LIN {X -0.012,Y -443.315,Z 1451.571,A 0.000,B 0.000,C 90.000,E1 282.715} C_DIS
LIN {X -0.002,Y -444.816,Z 1451.568,A 0.000,B 0.000,C 90.000,E1 282.187} C_DIS
LIN {X 0.020,Y -445.994,Z 1451.565,A 0.000,B 0.000,C 90.000,E1 281.658} C_DIS
LIN {X 0.049,Y -446.747,Z 1451.562,A 0.000,B 0.000,C 90.000,E1 281.130} C_DIS
LIN {X 0.083,Y -447.090,Z 1451.559,A 0.000,B 0.000,C 90.000,E1 280.602} C_DIS
LIN {X 0.118,Y -446.958,Z 1451.556,A 0.000,B 0.000,C 90.000,E1 280.074} C_DIS
LIN {X 0.078,Y -446.263,Z 1451.553,A 0.000,B 0.000,C 90.000,E1 279.557} C_DIS
LIN {X 0.112,Y -445.021,Z 1451.550,A 0.000,B 0.000,C 90.000,E1 279.029} C_DIS
LIN {X 0.071,Y -443.207,Z 1451.547,A 0.000,B 0.000,C 90.000,E1 278.511} C_DIS
LIN {X 0.025,Y -440.657,Z 1451.544,A 0.000,B 0.000,C 90.000,E1 277.992} C_DIS
LIN {X 0.022,Y -437.241,Z 1451.542,A 0.000,B 0.000,C 90.000,E1 277.466} C_DIS
LIN {X -0.056,Y -432.786,Z 1451.539,A 0.000,B 0.000,C 90.000,E1 276.947} C_DIS
LIN {X -0.155,Y -427.058,Z 1451.536,A 0.000,B 0.000,C 90.000,E1 276.429} C_DIS
LIN {X 0.194,Y -420.712,Z 1451.533,A 0.000,B 0.000,C 90.000,E1 275.910} C_DIS
LIN {X 0.170,Y -414.293,Z 1451.531,A 0.000,B 0.000,C 90.000,E1 275.511} C_DIS
LIN {X 0.133,Y -407.868,Z 1451.529,A 0.000,B 0.000,C 90.000,E1 275.163} C_DIS
LIN {X 0.107,Y -397.871,Z 1451.526,A 0.000,B 0.000,C 90.000,E1 274.702} C_DIS
LIN {X 0.086,Y -388.083,Z 1451.524,A 0.000,B 0.000,C 90.000,E1 274.302} C_DIS
LIN {X 0.003,Y -369.176,Z 1451.520,A 0.000,B 0.000,C 90.000,E1 273.612} C_DIS
LIN {X 0.038,Y -359.489,Z 1451.518,A 0.000,B 0.000,C 90.000,E1 273.269} C_DIS
LIN {X -0.062,Y -349.143,Z 1451.516,A 0.000,B 0.000,C 90.000,E1 272.980} C_DIS
LIN {X 0.134,Y -338.896,Z 1451.515,A 0.000,B 0.000,C 90.000,E1 272.694} C_DIS
LIN {X -0.136,Y -327.379,Z 1451.514,A 0.000,B 0.000,C 90.000,E1 272.522} C_DIS
LIN {X -0.109,Y -314.439,Z 1451.513,A 0.000,B 0.000,C 90.000,E1 272.350} C_DIS
LIN {X 0.000,Y -302.497,Z 1451.512,A 0.000,B 0.000,C 90.000,E1 272.236} C_DIS
LIN {X -0.035,Y -181.227,Z 1451.512,A 0.000,B 0.000,C 90.000,E1 272.236} C_DIS
LIN {X -0.026,Y -181.564,Z 1451.503,A 0.000,B 0.000,C 90.000,E1 270.516} C_DIS
LIN {X -0.036,Y -181.121,Z 1451.489,A 0.000,B 0.000,C 90.000,E1 267.993} C_DIS
LIN {X -0.047,Y -180.907,Z 1451.475,A 0.000,B 0.000,C 90.000,E1 265.469} C_DIS
LIN {X 0.009,Y -180.730,Z 1451.470,A 0.000,B 0.000,C 90.000,E1 264.609} C_DIS
LIN {X -0.069,Y -178.819,Z 1451.442,A 0.000,B 0.000,C 90.000,E1 259.567} C_DIS
LIN {X 0.013,Y -175.863,Z 1451.414,A 0.000,B 0.000,C 90.000,E1 254.448} C_DIS
LIN {X 0.062,Y -173.831,Z 1451.399,A 0.000,B 0.000,C 90.000,E1 251.873} C_DIS
LIN {X -0.003,Y -171.498,Z 1451.380,A 0.000,B 0.000,C 90.000,E1 248.465} C_DIS
LIN {X -0.017,Y -167.726,Z 1451.356,A 0.000,B 0.000,C 90.000,E1 244.152} C_DIS
LIN {X 0.000,Y -166.421,Z 1451.347,A 0.000,B 0.000,C 90.000,E1 242.410} C_DIS
LIN {X -0.002,Y -163.142,Z 1451.327,A 0.000,B 0.000,C 90.000,E1 238.918} C_DIS
LIN {X -0.036,Y -161.097,Z 1451.313,A 0.000,B 0.000,C 90.000,E1 236.294} C_DIS
LIN {X -0.052,Y -157.825,Z 1451.293,A 0.000,B 0.000,C 90.000,E1 232.763} C_DIS
LIN {X 0.011,Y -155.859,Z 1451.278,A 0.000,B 0.000,C 90.000,E1 230.070} C_DIS
LIN {X 0.067,Y -152.108,Z 1451.253,A 0.000,B 0.000,C 90.000,E1 225.567} C_DIS
LIN {X -0.026,Y -150.359,Z 1451.238,A 0.000,B 0.000,C 90.000,E1 222.894} C_DIS
LIN {X 0.013,Y -147.094,Z 1451.213,A 0.000,B 0.000,C 90.000,E1 218.338} C_DIS
LIN {X 0.008,Y -145.665,Z 1451.198,A 0.000,B 0.000,C 90.000,E1 215.598} C_DIS
LIN {X 0.012,Y -143.047,Z 1451.172,A 0.000,B 0.000,C 90.000,E1 211.003} C_DIS
LIN {X 0.012,Y -141.671,Z 1451.152,A 0.000,B 0.000,C 90.000,E1 207.308} C_DIS
LIN {X 0.057,Y -139.452,Z 1451.116,A 0.000,B 0.000,C 90.000,E1 200.791} C_DIS
LIN {X -0.023,Y -139.186,Z 1451.105,A 0.000,B 0.000,C 90.000,E1 198.960} C_DIS
LIN {X 0.000,Y -138.322,Z 1451.053,A 0.000,B 0.000,C 90.000,E1 189.613} C_DIS
LIN {X 0.007,Y -139.460,Z 1451.007,A 0.000,B 0.000,C 90.000,E1 181.203} C_DIS
LIN {X -0.053,Y -141.016,Z 1450.976,A 0.000,B 0.000,C 90.000,E1 175.641} C_DIS
LIN {X 0.037,Y -142.770,Z 1450.955,A 0.000,B 0.000,C 90.000,E1 171.894} C_DIS
LIN {X -0.007,Y -145.180,Z 1450.929,A 0.000,B 0.000,C 90.000,E1 167.297} C_DIS
LIN {X 0.026,Y -147.802,Z 1450.909,A 0.000,B 0.000,C 90.000,E1 163.614} C_DIS
LIN {X -0.079,Y -150.488,Z 1450.889,A 0.000,B 0.000,C 90.000,E1 160.007} C_DIS
LIN {X -0.007,Y -153.944,Z 1450.869,A 0.000,B 0.000,C 90.000,E1 156.357} C_DIS
LIN {X 0.057,Y -157.355,Z 1450.849,A 0.000,B 0.000,C 90.000,E1 152.743} C_DIS
LIN {X 0.000,Y -161.551,Z 1450.829,A 0.000,B 0.000,C 90.000,E1 149.203} C_DIS
LIN {X 0.013,Y -165.750,Z 1450.809,A 0.000,B 0.000,C 90.000,E1 145.674} C_DIS
LIN {X 0.000,Y -170.704,Z 1450.790,A 0.000,B 0.000,C 90.000,E1 142.190} C_DIS
LIN {X -0.089,Y -175.578,Z 1450.771,A 0.000,B 0.000,C 90.000,E1 138.771} C_DIS
LIN {X 0.030,Y -181.195,Z 1450.752,A 0.000,B 0.000,C 90.000,E1 135.324} C_DIS
LIN {X 0.023,Y -186.657,Z 1450.733,A 0.000,B 0.000,C 90.000,E1 131.962} C_DIS
LIN {X -0.032,Y -191.261,Z 1450.719,A 0.000,B 0.000,C 90.000,E1 129.483} C_DIS
LIN {X 0.048,Y -197.082,Z 1450.701,A 0.000,B 0.000,C 90.000,E1 126.171} C_DIS
LIN {X 0.036,Y -200.634,Z 1450.691,A 0.000,B 0.000,C 90.000,E1 124.405} C_DIS
LIN {X 0.020,Y -312.743,Z 1450.691,A 0.000,B 0.000,C 90.000,E1 124.405} C_DIS
LIN {X 0.046,Y -314.887,Z 1450.691,A 0.000,B 0.000,C 90.000,E1 124.358} C_DIS
LIN {X -0.085,Y -320.371,Z 1450.689,A 0.000,B 0.000,C 90.000,E1 124.072} C_DIS
LIN {X -0.040,Y -323.325,Z 1450.688,A 0.000,B 0.000,C 90.000,E1 123.754} C_DIS
LIN {X 0.032,Y -325.329,Z 1450.686,A 0.000,B 0.000,C 90.000,E1 123.452} C_DIS
LIN {X 0.015,Y -326.896,Z 1450.684,A 0.000,B 0.000,C 90.000,E1 123.166} C_DIS
LIN {X -0.061,Y -329.384,Z 1450.681,A 0.000,B 0.000,C 90.000,E1 122.546} C_DIS
LIN {X -0.136,Y -340.169,Z 1450.665,A 0.000,B 0.000,C 90.000,E1 119.745} C_DIS
LIN {X 0.067,Y -352.322,Z 1450.650,A 0.000,B 0.000,C 90.000,E1 116.950} C_DIS
LIN {X -0.017,Y -365.945,Z 1450.635,A 0.000,B 0.000,C 90.000,E1 114.259} C_DIS
LIN {X 0.042,Y -379.384,Z 1450.622,A 0.000,B 0.000,C 90.000,E1 111.897} C_DIS
LIN {X 0.170,Y -394.173,Z 1450.609,A 0.000,B 0.000,C 90.000,E1 109.577} C_DIS
LIN {X 0.040,Y -410.411,Z 1450.596,A 0.000,B 0.000,C 90.000,E1 107.347} C_DIS
LIN {X -0.222,Y -428.214,Z 1450.584,A 0.000,B 0.000,C 90.000,E1 105.190} C_DIS
LIN {X -0.210,Y -447.601,Z 1450.572,A 0.000,B 0.000,C 90.000,E1 103.063} C_DIS
LIN {X -0.068,Y -467.784,Z 1450.562,A 0.000,B 0.000,C 90.000,E1 101.074} C_DIS
LIN {X -0.089,Y -488.295,Z 1450.551,A 0.000,B 0.000,C 90.000,E1 99.265} C_DIS
LIN {X 0.066,Y -490.122,Z 1450.550,A 0.000,B 0.000,C 90.000,E1 99.029} C_DIS
LIN {X -0.110,Y -491.699,Z 1450.549,A 0.000,B 0.000,C 90.000,E1 98.803} C_DIS
LIN {X -0.211,Y -492.876,Z 1450.547,A 0.000,B 0.000,C 90.000,E1 98.568} C_DIS
LIN {X 0.020,Y -494.284,Z 1450.545,A 0.000,B 0.000,C 90.000,E1 98.049} C_DIS
LIN {X -0.229,Y -494.640,Z 1450.542,A 0.000,B 0.000,C 90.000,E1 97.587} C_DIS
LIN {X 0.022,Y -494.007,Z 1450.539,A 0.000,B 0.000,C 90.000,E1 97.068} C_DIS
LIN {X -0.215,Y -492.279,Z 1450.537,A 0.000,B 0.000,C 90.000,E1 96.606} C_DIS
LIN {X 0.180,Y -490.905,Z 1450.535,A 0.000,B 0.000,C 90.000,E1 96.315} C_DIS
LIN {X 0.168,Y -479.194,Z 1450.526,A 0.000,B 0.000,C 90.000,E1 94.588} C_DIS
LIN {X -0.108,Y -468.504,Z 1450.516,A 0.000,B 0.000,C 90.000,E1 92.865} C_DIS
LIN {X -0.173,Y -460.284,Z 1450.509,A 0.000,B 0.000,C 90.000,E1 91.604} C_DIS
LIN {X -0.173,Y -446.693,Z 1450.497,A 0.000,B 0.000,C 90.000,E1 89.542} C_DIS
LIN {X -0.032,Y -433.500,Z 1450.486,A 0.000,B 0.000,C 90.000,E1 87.421} C_DIS
LIN {X 0.123,Y -421.927,Z 1450.475,A 0.000,B 0.000,C 90.000,E1 85.527} C_DIS
LIN {X 0.073,Y -410.380,Z 1450.465,A 0.000,B 0.000,C 90.000,E1 83.628} C_DIS
LIN {X -0.173,Y -398.612,Z 1450.454,A 0.000,B 0.000,C 90.000,E1 81.724} C_DIS
LIN {X -0.138,Y -386.759,Z 1450.443,A 0.000,B 0.000,C 90.000,E1 79.746} C_DIS
LIN {X 0.106,Y -373.467,Z 1450.430,A 0.000,B 0.000,C 90.000,E1 77.409} C_DIS
LIN {X 0.123,Y -362.107,Z 1450.419,A 0.000,B 0.000,C 90.000,E1 75.353} C_DIS
LIN {X 0.085,Y -350.791,Z 1450.407,A 0.000,B 0.000,C 90.000,E1 73.268} C_DIS
LIN {X 0.017,Y -339.368,Z 1450.395,A 0.000,B 0.000,C 90.000,E1 71.148} C_DIS
LIN {X 0.116,Y -326.454,Z 1450.381,A 0.000,B 0.000,C 90.000,E1 68.646} C_DIS
LIN {X 0.065,Y -312.613,Z 1450.366,A 0.000,B 0.000,C 90.000,E1 65.793} C_DIS
LIN {X -0.090,Y -296.897,Z 1450.346,A 0.000,B 0.000,C 90.000,E1 62.231} C_DIS
LIN {X -0.034,Y -283.966,Z 1450.327,A 0.000,B 0.000,C 90.000,E1 58.869} C_DIS
LIN {X -0.109,Y -273.172,Z 1450.310,A 0.000,B 0.000,C 90.000,E1 55.801} C_DIS
LIN {X 0.034,Y -261.705,Z 1450.290,A 0.000,B 0.000,C 90.000,E1 52.271} C_DIS
LIN {X 0.069,Y -251.127,Z 1450.271,A 0.000,B 0.000,C 90.000,E1 48.690} C_DIS
LIN {X -0.076,Y -241.586,Z 1450.250,A 0.000,B 0.000,C 90.000,E1 45.081} C_DIS
LIN {X -0.007,Y -232.924,Z 1450.230,A 0.000,B 0.000,C 90.000,E1 41.353} C_DIS
LIN {X 0.022,Y -225.169,Z 1450.209,A 0.000,B 0.000,C 90.000,E1 37.569} C_DIS
LIN {X 0.120,Y -218.260,Z 1450.187,A 0.000,B 0.000,C 90.000,E1 33.706} C_DIS
LIN {X -0.101,Y -212.091,Z 1450.166,A 0.000,B 0.000,C 90.000,E1 29.873} C_DIS
LIN {X 0.016,Y -206.777,Z 1450.144,A 0.000,B 0.000,C 90.000,E1 25.899} C_DIS
LIN {X 0.071,Y -202.307,Z 1450.122,A 0.000,B 0.000,C 90.000,E1 21.897} C_DIS
LIN {X -0.033,Y -197.929,Z 1450.095,A 0.000,B 0.000,C 90.000,E1 17.094} C_DIS
LIN {X 0.071,Y -194.655,Z 1450.068,A 0.000,B 0.000,C 90.000,E1 12.187} C_DIS
LIN {X 0.043,Y -192.713,Z 1450.045,A 0.000,B 0.000,C 90.000,E1 8.106} C_DIS
LIN {X 0.053,Y -190.911,Z 1450.013,A 0.000,B 0.000,C 90.000,E1 2.350} C_DIS
LIN {X 0.010,Y -190.278,Z 1449.988,A 0.000,B 0.000,C 90.000,E1 357.879} C_DIS
LIN {X -0.079,Y -190.435,Z 1449.956,A 0.000,B 0.000,C 90.000,E1 352.129} C_DIS
LIN {X -0.059,Y -191.810,Z 1449.924,A 0.000,B 0.000,C 90.000,E1 346.353} C_DIS
LIN {X -0.056,Y -194.696,Z 1449.892,A 0.000,B 0.000,C 90.000,E1 340.604} C_DIS
LIN {X 0.105,Y -198.511,Z 1449.865,A 0.000,B 0.000,C 90.000,E1 335.665} C_DIS
LIN {X 0.039,Y -202.895,Z 1449.843,A 0.000,B 0.000,C 90.000,E1 331.641} C_DIS
LIN {X -0.042,Y -208.476,Z 1449.820,A 0.000,B 0.000,C 90.000,E1 327.661} C_DIS
LIN {X 0.003,Y -213.898,Z 1449.803,A 0.000,B 0.000,C 90.000,E1 324.482} C_DIS
LIN {X 0.088,Y -220.301,Z 1449.785,A 0.000,B 0.000,C 90.000,E1 321.331} C_DIS
LIN {X 0.039,Y -228.594,Z 1449.766,A 0.000,B 0.000,C 90.000,E1 317.877} C_DIS
LIN {X -0.120,Y -238.107,Z 1449.747,A 0.000,B 0.000,C 90.000,E1 314.514} C_DIS
LIN {X 0.017,Y -247.599,Z 1449.731,A 0.000,B 0.000,C 90.000,E1 311.515} C_DIS
LIN {X -0.026,Y -259.668,Z 1449.713,A 0.000,B 0.000,C 90.000,E1 308.257} C_DIS
LIN {X 0.028,Y -270.155,Z 1449.699,A 0.000,B 0.000,C 90.000,E1 305.758} C_DIS
LIN {X 0.067,Y -280.287,Z 1449.687,A 0.000,B 0.000,C 90.000,E1 303.658} C_DIS
LIN {X 0.017,Y -289.691,Z 1449.678,A 0.000,B 0.000,C 90.000,E1 301.957} C_DIS
LIN {X 0.108,Y -300.162,Z 1449.668,A 0.000,B 0.000,C 90.000,E1 300.256} C_DIS
LIN {X 0.028,Y -309.441,Z 1449.661,A 0.000,B 0.000,C 90.000,E1 298.949} C_DIS
LIN {X -0.048,Y -319.596,Z 1449.654,A 0.000,B 0.000,C 90.000,E1 297.692} C_DIS
LIN {X -0.052,Y -335.747,Z 1449.644,A 0.000,B 0.000,C 90.000,E1 295.899} C_DIS
LIN {X -0.142,Y -349.504,Z 1449.636,A 0.000,B 0.000,C 90.000,E1 294.515} C_DIS
LIN {X 0.040,Y -362.886,Z 1449.629,A 0.000,B 0.000,C 90.000,E1 293.131} C_DIS
LIN {X -0.080,Y -373.257,Z 1449.623,A 0.000,B 0.000,C 90.000,E1 292.078} C_DIS
LIN {X 0.040,Y -386.282,Z 1449.615,A 0.000,B 0.000,C 90.000,E1 290.663} C_DIS
LIN {X -0.199,Y -396.420,Z 1449.609,A 0.000,B 0.000,C 90.000,E1 289.577} C_DIS
LIN {X 0.146,Y -408.840,Z 1449.601,A 0.000,B 0.000,C 90.000,E1 288.127} C_DIS
LIN {X -0.081,Y -416.029,Z 1449.596,A 0.000,B 0.000,C 90.000,E1 287.330} C_DIS
LIN {X 0.001,Y -422.783,Z 1449.592,A 0.000,B 0.000,C 90.000,E1 286.496} C_DIS
LIN {X 0.155,Y -428.836,Z 1449.587,A 0.000,B 0.000,C 90.000,E1 285.662} C_DIS
LIN {X -0.168,Y -433.987,Z 1449.583,A 0.000,B 0.000,C 90.000,E1 284.898} C_DIS
LIN {X 0.092,Y -438.179,Z 1449.578,A 0.000,B 0.000,C 90.000,E1 284.064} C_DIS
LIN {X 0.074,Y -440.546,Z 1449.575,A 0.000,B 0.000,C 90.000,E1 283.536} C_DIS
LIN {X -0.143,Y -443.448,Z 1449.571,A 0.000,B 0.000,C 90.000,E1 282.771} C_DIS
LIN {X -0.133,Y -444.982,Z 1449.568,A 0.000,B 0.000,C 90.000,E1 282.243} C_DIS
LIN {X -0.112,Y -446.197,Z 1449.565,A 0.000,B 0.000,C 90.000,E1 281.715} C_DIS
LIN {X -0.083,Y -447.028,Z 1449.562,A 0.000,B 0.000,C 90.000,E1 281.186} C_DIS
LIN {X -0.049,Y -447.415,Z 1449.559,A 0.000,B 0.000,C 90.000,E1 280.658} C_DIS
LIN {X -0.092,Y -447.295,Z 1449.556,A 0.000,B 0.000,C 90.000,E1 280.141} C_DIS
LIN {X -0.052,Y -446.719,Z 1449.553,A 0.000,B 0.000,C 90.000,E1 279.613} C_DIS
LIN {X -0.087,Y -445.545,Z 1449.550,A 0.000,B 0.000,C 90.000,E1 279.095} C_DIS
LIN {X -0.055,Y -443.776,Z 1449.548,A 0.000,B 0.000,C 90.000,E1 278.568} C_DIS
LIN {X -0.097,Y -441.304,Z 1449.545,A 0.000,B 0.000,C 90.000,E1 278.049} C_DIS
LIN {X -0.153,Y -437.981,Z 1449.542,A 0.000,B 0.000,C 90.000,E1 277.530} C_DIS
LIN {X -0.170,Y -433.708,Z 1449.539,A 0.000,B 0.000,C 90.000,E1 277.004} C_DIS
LIN {X 0.163,Y -428.146,Z 1449.536,A 0.000,B 0.000,C 90.000,E1 276.429} C_DIS
LIN {X -0.017,Y -421.798,Z 1449.533,A 0.000,B 0.000,C 90.000,E1 275.967} C_DIS
LIN {X -0.118,Y -415.309,Z 1449.531,A 0.000,B 0.000,C 90.000,E1 275.568} C_DIS
LIN {X -0.198,Y -408.819,Z 1449.529,A 0.000,B 0.000,C 90.000,E1 275.220} C_DIS
LIN {X -0.046,Y -402.223,Z 1449.527,A 0.000,B 0.000,C 90.000,E1 274.878} C_DIS
LIN {X -0.152,Y -392.450,Z 1449.525,A 0.000,B 0.000,C 90.000,E1 274.473} C_DIS
LIN {X 0.004,Y -379.550,Z 1449.522,A 0.000,B 0.000,C 90.000,E1 273.955} C_DIS
LIN {X 0.027,Y -363.639,Z 1449.519,A 0.000,B 0.000,C 90.000,E1 273.383} C_DIS
LIN {X -0.123,Y -353.816,Z 1449.517,A 0.000,B 0.000,C 90.000,E1 273.094} C_DIS
LIN {X 0.163,Y -339.985,Z 1449.515,A 0.000,B 0.000,C 90.000,E1 272.694} C_DIS
LIN {X -0.039,Y -332.780,Z 1449.514,A 0.000,B 0.000,C 90.000,E1 272.579} C_DIS
LIN {X -0.099,Y -320.374,Z 1449.513,A 0.000,B 0.000,C 90.000,E1 272.407} C_DIS
LIN {X -0.029,Y -310.790,Z 1449.513,A 0.000,B 0.000,C 90.000,E1 272.293} C_DIS
LIN {X -0.021,Y -301.329,Z 1449.512,A 0.000,B 0.000,C 90.000,E1 272.236} C_DIS
LIN {X -0.048,Y -181.227,Z 1449.512,A 0.000,B 0.000,C 90.000,E1 272.236} C_DIS
LIN {X -0.007,Y -181.563,Z 1449.503,A 0.000,B 0.000,C 90.000,E1 270.516} C_DIS
LIN {X -0.077,Y -181.281,Z 1449.494,A 0.000,B 0.000,C 90.000,E1 268.854} C_DIS
LIN {X -0.028,Y -180.906,Z 1449.475,A 0.000,B 0.000,C 90.000,E1 265.469} C_DIS
LIN {X 0.029,Y -180.733,Z 1449.470,A 0.000,B 0.000,C 90.000,E1 264.609} C_DIS
LIN {X -0.050,Y -178.821,Z 1449.442,A 0.000,B 0.000,C 90.000,E1 259.567} C_DIS
LIN {X 0.032,Y -175.866,Z 1449.414,A 0.000,B 0.000,C 90.000,E1 254.448} C_DIS
LIN {X 0.027,Y -173.835,Z 1449.399,A 0.000,B 0.000,C 90.000,E1 251.891} C_DIS
LIN {X 0.016,Y -171.504,Z 1449.380,A 0.000,B 0.000,C 90.000,E1 248.465} C_DIS
LIN {X 0.003,Y -167.731,Z 1449.356,A 0.000,B 0.000,C 90.000,E1 244.152} C_DIS
LIN {X 0.018,Y -166.427,Z 1449.347,A 0.000,B 0.000,C 90.000,E1 242.410} C_DIS
LIN {X 0.016,Y -163.148,Z 1449.327,A 0.000,B 0.000,C 90.000,E1 238.918} C_DIS
LIN {X -0.018,Y -161.103,Z 1449.313,A 0.000,B 0.000,C 90.000,E1 236.294} C_DIS
LIN {X -0.035,Y -157.830,Z 1449.293,A 0.000,B 0.000,C 90.000,E1 232.763} C_DIS
LIN {X 0.029,Y -155.864,Z 1449.278,A 0.000,B 0.000,C 90.000,E1 230.070} C_DIS
LIN {X 0.084,Y -152.113,Z 1449.253,A 0.000,B 0.000,C 90.000,E1 225.567} C_DIS
LIN {X -0.008,Y -150.363,Z 1449.238,A 0.000,B 0.000,C 90.000,E1 222.894} C_DIS
LIN {X 0.030,Y -147.099,Z 1449.213,A 0.000,B 0.000,C 90.000,E1 218.338} C_DIS
LIN {X 0.025,Y -145.668,Z 1449.198,A 0.000,B 0.000,C 90.000,E1 215.598} C_DIS
LIN {X 0.028,Y -143.051,Z 1449.172,A 0.000,B 0.000,C 90.000,E1 211.003} C_DIS
LIN {X -0.036,Y -141.673,Z 1449.152,A 0.000,B 0.000,C 90.000,E1 207.334} C_DIS
LIN {X 0.072,Y -139.453,Z 1449.116,A 0.000,B 0.000,C 90.000,E1 200.791} C_DIS
LIN {X -0.007,Y -139.187,Z 1449.105,A 0.000,B 0.000,C 90.000,E1 198.960} C_DIS
LIN {X 0.016,Y -138.322,Z 1449.053,A 0.000,B 0.000,C 90.000,E1 189.613} C_DIS
LIN {X 0.023,Y -139.459,Z 1449.007,A 0.000,B 0.000,C 90.000,E1 181.203} C_DIS
LIN {X -0.036,Y -141.013,Z 1448.976,A 0.000,B 0.000,C 90.000,E1 175.641} C_DIS
LIN {X 0.054,Y -142.767,Z 1448.955,A 0.000,B 0.000,C 90.000,E1 171.894} C_DIS
LIN {X 0.009,Y -145.176,Z 1448.929,A 0.000,B 0.000,C 90.000,E1 167.297} C_DIS
LIN {X 0.042,Y -147.798,Z 1448.909,A 0.000,B 0.000,C 90.000,E1 163.614} C_DIS
LIN {X -0.062,Y -150.482,Z 1448.889,A 0.000,B 0.000,C 90.000,E1 160.007} C_DIS
LIN {X 0.011,Y -153.937,Z 1448.869,A 0.000,B 0.000,C 90.000,E1 156.357} C_DIS
LIN {X 0.075,Y -157.348,Z 1448.849,A 0.000,B 0.000,C 90.000,E1 152.743} C_DIS
LIN {X 0.018,Y -161.543,Z 1448.829,A 0.000,B 0.000,C 90.000,E1 149.203} C_DIS
LIN {X 0.030,Y -165.742,Z 1448.809,A 0.000,B 0.000,C 90.000,E1 145.674} C_DIS
LIN {X 0.018,Y -170.694,Z 1448.790,A 0.000,B 0.000,C 90.000,E1 142.190} C_DIS
LIN {X -0.071,Y -175.568,Z 1448.771,A 0.000,B 0.000,C 90.000,E1 138.771} C_DIS
LIN {X 0.049,Y -181.186,Z 1448.752,A 0.000,B 0.000,C 90.000,E1 135.324} C_DIS
LIN {X -0.082,Y -186.646,Z 1448.733,A 0.000,B 0.000,C 90.000,E1 132.000} C_DIS
LIN {X -0.013,Y -191.252,Z 1448.719,A 0.000,B 0.000,C 90.000,E1 129.483} C_DIS
LIN {X 0.068,Y -197.071,Z 1448.701,A 0.000,B 0.000,C 90.000,E1 126.171} C_DIS
LIN {X -0.031,Y -200.580,Z 1448.691,A 0.000,B 0.000,C 90.000,E1 124.452} C_DIS
LIN {X 0.158,Y -312.400,Z 1448.691,A 0.000,B 0.000,C 90.000,E1 124.405} C_DIS
LIN {X -0.080,Y -317.681,Z 1448.690,A 0.000,B 0.000,C 90.000,E1 124.278} C_DIS
LIN {X -0.144,Y -320.108,Z 1448.689,A 0.000,B 0.000,C 90.000,E1 124.119} C_DIS
LIN {X -0.188,Y -323.361,Z 1448.688,A 0.000,B 0.000,C 90.000,E1 123.785} C_DIS
LIN {X 0.066,Y -325.332,Z 1448.686,A 0.000,B 0.000,C 90.000,E1 123.452} C_DIS
LIN {X 0.049,Y -326.878,Z 1448.684,A 0.000,B 0.000,C 90.000,E1 123.166} C_DIS
LIN {X -0.025,Y -329.341,Z 1448.681,A 0.000,B 0.000,C 90.000,E1 122.546} C_DIS
LIN {X -0.102,Y -340.123,Z 1448.665,A 0.000,B 0.000,C 90.000,E1 119.745} C_DIS
LIN {X 0.101,Y -352.275,Z 1448.650,A 0.000,B 0.000,C 90.000,E1 116.950} C_DIS
LIN {X 0.017,Y -365.892,Z 1448.635,A 0.000,B 0.000,C 90.000,E1 114.259} C_DIS
LIN {X 0.076,Y -379.329,Z 1448.622,A 0.000,B 0.000,C 90.000,E1 111.897} C_DIS
LIN {X -0.168,Y -394.114,Z 1448.609,A 0.000,B 0.000,C 90.000,E1 109.631} C_DIS
LIN {X 0.074,Y -410.349,Z 1448.596,A 0.000,B 0.000,C 90.000,E1 107.347} C_DIS
LIN {X -0.188,Y -428.149,Z 1448.584,A 0.000,B 0.000,C 90.000,E1 105.190} C_DIS
LIN {X -0.176,Y -447.532,Z 1448.572,A 0.000,B 0.000,C 90.000,E1 103.063} C_DIS
LIN {X -0.037,Y -467.715,Z 1448.562,A 0.000,B 0.000,C 90.000,E1 101.074} C_DIS
LIN {X -0.216,Y -485.820,Z 1448.553,A 0.000,B 0.000,C 90.000,E1 99.500} C_DIS
LIN {X -0.061,Y -488.216,Z 1448.551,A 0.000,B 0.000,C 90.000,E1 99.265} C_DIS
LIN {X 0.094,Y -490.036,Z 1448.550,A 0.000,B 0.000,C 90.000,E1 99.029} C_DIS
LIN {X -0.082,Y -491.607,Z 1448.549,A 0.000,B 0.000,C 90.000,E1 98.803} C_DIS
LIN {X -0.183,Y -492.779,Z 1448.547,A 0.000,B 0.000,C 90.000,E1 98.568} C_DIS
LIN {X 0.048,Y -494.181,Z 1448.545,A 0.000,B 0.000,C 90.000,E1 98.049} C_DIS
LIN {X -0.201,Y -494.532,Z 1448.542,A 0.000,B 0.000,C 90.000,E1 97.587} C_DIS
LIN {X 0.048,Y -493.891,Z 1448.539,A 0.000,B 0.000,C 90.000,E1 97.068} C_DIS
LIN {X -0.189,Y -492.157,Z 1448.537,A 0.000,B 0.000,C 90.000,E1 96.606} C_DIS
LIN {X 0.206,Y -490.779,Z 1448.535,A 0.000,B 0.000,C 90.000,E1 96.315} C_DIS
LIN {X 0.190,Y -479.064,Z 1448.526,A 0.000,B 0.000,C 90.000,E1 94.588} C_DIS
LIN {X -0.090,Y -468.330,Z 1448.516,A 0.000,B 0.000,C 90.000,E1 92.865} C_DIS
LIN {X -0.156,Y -460.116,Z 1448.509,A 0.000,B 0.000,C 90.000,E1 91.604} C_DIS
LIN {X -0.161,Y -446.531,Z 1448.497,A 0.000,B 0.000,C 90.000,E1 89.542} C_DIS
LIN {X -0.023,Y -433.380,Z 1448.486,A 0.000,B 0.000,C 90.000,E1 87.421} C_DIS
LIN {X 0.128,Y -421.841,Z 1448.475,A 0.000,B 0.000,C 90.000,E1 85.527} C_DIS
LIN {X 0.077,Y -410.317,Z 1448.465,A 0.000,B 0.000,C 90.000,E1 83.628} C_DIS
LIN {X 0.197,Y -400.277,Z 1448.455,A 0.000,B 0.000,C 90.000,E1 81.951} C_DIS
LIN {X 0.136,Y -390.147,Z 1448.446,A 0.000,B 0.000,C 90.000,E1 80.274} C_DIS
LIN {X 0.095,Y -375.153,Z 1448.432,A 0.000,B 0.000,C 90.000,E1 77.701} C_DIS
LIN {X 0.126,Y -362.153,Z 1448.419,A 0.000,B 0.000,C 90.000,E1 75.353} C_DIS
LIN {X 0.089,Y -350.841,Z 1448.407,A 0.000,B 0.000,C 90.000,E1 73.268} C_DIS
LIN {X 0.023,Y -339.397,Z 1448.395,A 0.000,B 0.000,C 90.000,E1 71.148} C_DIS
LIN {X 0.091,Y -324.893,Z 1448.380,A 0.000,B 0.000,C 90.000,E1 68.337} C_DIS
LIN {X 0.042,Y -309.587,Z 1448.362,A 0.000,B 0.000,C 90.000,E1 65.153} C_DIS
LIN {X -0.067,Y -294.164,Z 1448.342,A 0.000,B 0.000,C 90.000,E1 61.563} C_DIS
LIN {X -0.091,Y -281.508,Z 1448.323,A 0.000,B 0.000,C 90.000,E1 58.201} C_DIS
LIN {X -0.080,Y -270.840,Z 1448.306,A 0.000,B 0.000,C 90.000,E1 55.102} C_DIS
LIN {X 0.146,Y -259.551,Z 1448.286,A 0.000,B 0.000,C 90.000,E1 51.537} C_DIS
LIN {X -0.071,Y -249.245,Z 1448.267,A 0.000,B 0.000,C 90.000,E1 48.000} C_DIS
LIN {X -0.101,Y -239.895,Z 1448.246,A 0.000,B 0.000,C 90.000,E1 44.352} C_DIS
LIN {X -0.068,Y -231.430,Z 1448.226,A 0.000,B 0.000,C 90.000,E1 40.620} C_DIS
LIN {X 0.098,Y -223.864,Z 1448.204,A 0.000,B 0.000,C 90.000,E1 36.790} C_DIS
LIN {X 0.033,Y -217.119,Z 1448.183,A 0.000,B 0.000,C 90.000,E1 32.959} C_DIS
LIN {X -0.037,Y -211.140,Z 1448.161,A 0.000,B 0.000,C 90.000,E1 29.077} C_DIS
LIN {X 0.049,Y -206.007,Z 1448.140,A 0.000,B 0.000,C 90.000,E1 25.103} C_DIS
LIN {X 0.089,Y -201.717,Z 1448.117,A 0.000,B 0.000,C 90.000,E1 21.099} C_DIS
LIN {X 0.089,Y -197.538,Z 1448.090,A 0.000,B 0.000,C 90.000,E1 16.260} C_DIS
LIN {X -0.043,Y -194.077,Z 1448.059,A 0.000,B 0.000,C 90.000,E1 10.602} C_DIS
LIN {X -0.026,Y -192.080,Z 1448.031,A 0.000,B 0.000,C 90.000,E1 5.682} C_DIS
LIN {X 0.000,Y -190.781,Z 1448.000,A 0.000,B 0.000,C 90.000,E1 360.000} C_DIS
LIN {X 0.057,Y -190.548,Z 1447.965,A 0.000,B 0.000,C 90.000,E1 353.742} C_DIS
LIN {X -0.014,Y -191.511,Z 1447.933,A 0.000,B 0.000,C 90.000,E1 347.993} C_DIS
LIN {X 0.050,Y -194.359,Z 1447.897,A 0.000,B 0.000,C 90.000,E1 341.402} C_DIS
LIN {X -0.063,Y -197.940,Z 1447.870,A 0.000,B 0.000,C 90.000,E1 336.538} C_DIS
LIN {X -0.058,Y -202.083,Z 1447.847,A 0.000,B 0.000,C 90.000,E1 332.487} C_DIS
LIN {X 0.015,Y -207.412,Z 1447.825,A 0.000,B 0.000,C 90.000,E1 328.456} C_DIS
LIN {X -0.081,Y -212.598,Z 1447.807,A 0.000,B 0.000,C 90.000,E1 325.308} C_DIS
LIN {X 0.015,Y -218.760,Z 1447.790,A 0.000,B 0.000,C 90.000,E1 322.145} C_DIS
LIN {X -0.015,Y -225.855,Z 1447.772,A 0.000,B 0.000,C 90.000,E1 319.057} C_DIS
LIN {X 0.132,Y -233.915,Z 1447.756,A 0.000,B 0.000,C 90.000,E1 315.972} C_DIS
LIN {X -0.004,Y -242.872,Z 1447.739,A 0.000,B 0.000,C 90.000,E1 313.014} C_DIS
LIN {X -0.069,Y -252.942,Z 1447.723,A 0.000,B 0.000,C 90.000,E1 310.092} C_DIS
LIN {X -0.015,Y -264.164,Z 1447.707,A 0.000,B 0.000,C 90.000,E1 307.202} C_DIS
LIN {X -0.022,Y -271.886,Z 1447.697,A 0.000,B 0.000,C 90.000,E1 305.438} C_DIS
LIN {X -0.116,Y -282.187,Z 1447.685,A 0.000,B 0.000,C 90.000,E1 303.372} C_DIS
LIN {X -0.151,Y -291.771,Z 1447.676,A 0.000,B 0.000,C 90.000,E1 301.671} C_DIS
LIN {X 0.080,Y -302.423,Z 1447.667,A 0.000,B 0.000,C 90.000,E1 299.951} C_DIS
LIN {X 0.183,Y -311.964,Z 1447.659,A 0.000,B 0.000,C 90.000,E1 298.615} C_DIS
LIN {X 0.103,Y -322.205,Z 1447.652,A 0.000,B 0.000,C 90.000,E1 297.385} C_DIS
LIN {X 0.013,Y -335.628,Z 1447.644,A 0.000,B 0.000,C 90.000,E1 295.924} C_DIS
LIN {X 0.050,Y -351.966,Z 1447.635,A 0.000,B 0.000,C 90.000,E1 294.259} C_DIS
LIN {X 0.019,Y -365.399,Z 1447.627,A 0.000,B 0.000,C 90.000,E1 292.898} C_DIS
LIN {X 0.014,Y -373.287,Z 1447.623,A 0.000,B 0.000,C 90.000,E1 292.078} C_DIS
LIN {X 0.136,Y -386.290,Z 1447.615,A 0.000,B 0.000,C 90.000,E1 290.663} C_DIS
LIN {X 0.222,Y -393.905,Z 1447.610,A 0.000,B 0.000,C 90.000,E1 289.812} C_DIS
LIN {X 0.147,Y -406.400,Z 1447.602,A 0.000,B 0.000,C 90.000,E1 288.417} C_DIS
LIN {X -0.021,Y -416.104,Z 1447.596,A 0.000,B 0.000,C 90.000,E1 287.330} C_DIS
LIN {X 0.062,Y -422.914,Z 1447.592,A 0.000,B 0.000,C 90.000,E1 286.496} C_DIS
LIN {X 0.220,Y -428.984,Z 1447.587,A 0.000,B 0.000,C 90.000,E1 285.662} C_DIS
LIN {X -0.101,Y -434.154,Z 1447.583,A 0.000,B 0.000,C 90.000,E1 284.898} C_DIS
LIN {X 0.160,Y -438.400,Z 1447.578,A 0.000,B 0.000,C 90.000,E1 284.064} C_DIS
LIN {X -0.076,Y -441.796,Z 1447.574,A 0.000,B 0.000,C 90.000,E1 283.300} C_DIS
LIN {X -0.071,Y -443.669,Z 1447.571,A 0.000,B 0.000,C 90.000,E1 282.771} C_DIS
LIN {X -0.059,Y -445.226,Z 1447.568,A 0.000,B 0.000,C 90.000,E1 282.243} C_DIS
LIN {X -0.037,Y -446.431,Z 1447.565,A 0.000,B 0.000,C 90.000,E1 281.715} C_DIS
LIN {X -0.007,Y -447.299,Z 1447.562,A 0.000,B 0.000,C 90.000,E1 281.186} C_DIS
LIN {X 0.029,Y -447.702,Z 1447.559,A 0.000,B 0.000,C 90.000,E1 280.658} C_DIS
LIN {X -0.011,Y -447.640,Z 1447.556,A 0.000,B 0.000,C 90.000,E1 280.141} C_DIS
LIN {X 0.030,Y -447.079,Z 1447.553,A 0.000,B 0.000,C 90.000,E1 279.613} C_DIS
LIN {X -0.003,Y -445.940,Z 1447.551,A 0.000,B 0.000,C 90.000,E1 279.095} C_DIS
LIN {X 0.031,Y -444.218,Z 1447.548,A 0.000,B 0.000,C 90.000,E1 278.568} C_DIS
LIN {X -0.010,Y -441.769,Z 1447.545,A 0.000,B 0.000,C 90.000,E1 278.049} C_DIS
LIN {X 0.210,Y -440.265,Z 1447.543,A 0.000,B 0.000,C 90.000,E1 277.757} C_DIS
LIN {X 0.146,Y -436.521,Z 1447.540,A 0.000,B 0.000,C 90.000,E1 277.239} C_DIS
LIN {X -0.079,Y -434.295,Z 1447.539,A 0.000,B 0.000,C 90.000,E1 277.004} C_DIS
LIN {X -0.170,Y -428.853,Z 1447.536,A 0.000,B 0.000,C 90.000,E1 276.486} C_DIS
LIN {X 0.048,Y -422.546,Z 1447.533,A 0.000,B 0.000,C 90.000,E1 275.967} C_DIS
LIN {X -0.082,Y -416.082,Z 1447.531,A 0.000,B 0.000,C 90.000,E1 275.568} C_DIS
LIN {X -0.167,Y -409.672,Z 1447.529,A 0.000,B 0.000,C 90.000,E1 275.220} C_DIS
LIN {X 0.201,Y -399.917,Z 1447.526,A 0.000,B 0.000,C 90.000,E1 274.702} C_DIS
LIN {X 0.134,Y -390.198,Z 1447.524,A 0.000,B 0.000,C 90.000,E1 274.302} C_DIS
LIN {X -0.050,Y -374.061,Z 1447.521,A 0.000,B 0.000,C 90.000,E1 273.726} C_DIS
LIN {X 0.052,Y -361.285,Z 1447.518,A 0.000,B 0.000,C 90.000,E1 273.269} C_DIS
LIN {X -0.035,Y -351.071,Z 1447.516,A 0.000,B 0.000,C 90.000,E1 272.980} C_DIS
LIN {X 0.072,Y -337.517,Z 1447.515,A 0.000,B 0.000,C 90.000,E1 272.636} C_DIS
LIN {X -0.086,Y -325.804,Z 1447.514,A 0.000,B 0.000,C 90.000,E1 272.465} C_DIS
LIN {X 0.024,Y -312.494,Z 1447.513,A 0.000,B 0.000,C 90.000,E1 272.293} C_DIS
LIN {X -0.024,Y -300.897,Z 1447.512,A 0.000,B 0.000,C 90.000,E1 272.236} C_DIS
LIN {X -0.050,Y -181.227,Z 1447.512,A 0.000,B 0.000,C 90.000,E1 272.236} C_DIS
LIN {X 0.052,Y -181.579,Z 1447.501,A 0.000,B 0.000,C 90.000,E1 270.172} C_DIS
LIN {X 0.041,Y -180.888,Z 1447.473,A 0.000,B 0.000,C 90.000,E1 265.122} C_DIS
LIN {X -0.076,Y -179.009,Z 1447.445,A 0.000,B 0.000,C 90.000,E1 260.095} C_DIS
LIN {X 0.019,Y -178.624,Z 1447.440,A 0.000,B 0.000,C 90.000,E1 259.218} C_DIS
LIN {X -0.083,Y -175.675,Z 1447.412,A 0.000,B 0.000,C 90.000,E1 254.157} C_DIS
LIN {X -0.071,Y -172.392,Z 1447.388,A 0.000,B 0.000,C 90.000,E1 249.880} C_DIS
LIN {X -0.055,Y -171.197,Z 1447.379,A 0.000,B 0.000,C 90.000,E1 248.156} C_DIS
LIN {X -0.003,Y -167.486,Z 1447.354,A 0.000,B 0.000,C 90.000,E1 243.819} C_DIS
LIN {X 0.005,Y -166.882,Z 1447.350,A 0.000,B 0.000,C 90.000,E1 242.948} C_DIS
LIN {X -0.004,Y -162.188,Z 1447.321,A 0.000,B 0.000,C 90.000,E1 237.709} C_DIS
LIN {X -0.036,Y -160.757,Z 1447.311,A 0.000,B 0.000,C 90.000,E1 235.960} C_DIS
LIN {X 0.031,Y -157.555,Z 1447.291,A 0.000,B 0.000,C 90.000,E1 232.396} C_DIS
LIN {X -0.030,Y -155.583,Z 1447.276,A 0.000,B 0.000,C 90.000,E1 229.747} C_DIS
LIN {X 0.022,Y -151.868,Z 1447.251,A 0.000,B 0.000,C 90.000,E1 225.243} C_DIS
LIN {X 0.035,Y -150.092,Z 1447.236,A 0.000,B 0.000,C 90.000,E1 222.528} C_DIS
LIN {X -0.047,Y -146.892,Z 1447.211,A 0.000,B 0.000,C 90.000,E1 218.016} C_DIS
LIN {X 0.056,Y -145.479,Z 1447.196,A 0.000,B 0.000,C 90.000,E1 215.231} C_DIS
LIN {X -0.026,Y -142.889,Z 1447.170,A 0.000,B 0.000,C 90.000,E1 210.669} C_DIS
LIN {X 0.031,Y -141.508,Z 1447.150,A 0.000,B 0.000,C 90.000,E1 206.950} C_DIS
LIN {X -0.052,Y -139.391,Z 1447.114,A 0.000,B 0.000,C 90.000,E1 200.482} C_DIS
LIN {X -0.001,Y -139.098,Z 1447.103,A 0.000,B 0.000,C 90.000,E1 198.598} C_DIS
LIN {X -0.009,Y -138.354,Z 1447.057,A 0.000,B 0.000,C 90.000,E1 190.197} C_DIS
LIN {X -0.016,Y -139.514,Z 1447.005,A 0.000,B 0.000,C 90.000,E1 180.859} C_DIS
LIN {X 0.065,Y -141.166,Z 1446.974,A 0.000,B 0.000,C 90.000,E1 175.241} C_DIS
LIN {X 0.036,Y -142.546,Z 1446.958,A 0.000,B 0.000,C 90.000,E1 172.470} C_DIS
LIN {X -0.037,Y -144.820,Z 1446.933,A 0.000,B 0.000,C 90.000,E1 167.881} C_DIS
LIN {X -0.051,Y -147.441,Z 1446.912,A 0.000,B 0.000,C 90.000,E1 164.212} C_DIS
LIN {X -0.023,Y -150.022,Z 1446.892,A 0.000,B 0.000,C 90.000,E1 160.550} C_DIS
LIN {X -0.016,Y -153.357,Z 1446.872,A 0.000,B 0.000,C 90.000,E1 156.922} C_DIS
LIN {X 0.033,Y -155.890,Z 1446.857,A 0.000,B 0.000,C 90.000,E1 154.204} C_DIS
LIN {X -0.069,Y -159.748,Z 1446.837,A 0.000,B 0.000,C 90.000,E1 150.667} C_DIS
LIN {X -0.004,Y -161.988,Z 1446.827,A 0.000,B 0.000,C 90.000,E1 148.869} C_DIS
LIN {X 0.016,Y -166.180,Z 1446.807,A 0.000,B 0.000,C 90.000,E1 145.341} C_DIS
LIN {X 0.009,Y -171.195,Z 1446.788,A 0.000,B 0.000,C 90.000,E1 141.859} C_DIS
LIN {X 0.039,Y -176.078,Z 1446.769,A 0.000,B 0.000,C 90.000,E1 138.405} C_DIS
LIN {X -0.099,Y -180.337,Z 1446.755,A 0.000,B 0.000,C 90.000,E1 135.891} C_DIS
LIN {X 0.009,Y -185.747,Z 1446.736,A 0.000,B 0.000,C 90.000,E1 132.486} C_DIS
LIN {X -0.077,Y -190.358,Z 1446.722,A 0.000,B 0.000,C 90.000,E1 130.011} C_DIS
LIN {X -0.031,Y -197.684,Z 1446.699,A 0.000,B 0.000,C 90.000,E1 125.884} C_DIS
LIN {X -0.064,Y -200.535,Z 1446.692,A 0.000,B 0.000,C 90.000,E1 124.485} C_DIS
LIN {X 0.040,Y -312.022,Z 1446.691,A 0.000,B 0.000,C 90.000,E1 124.452} C_DIS
LIN {X 0.018,Y -318.207,Z 1446.690,A 0.000,B 0.000,C 90.000,E1 124.246} C_DIS
LIN {X -0.025,Y -320.920,Z 1446.689,A 0.000,B 0.000,C 90.000,E1 124.040} C_DIS
LIN {X -0.034,Y -324.693,Z 1446.687,A 0.000,B 0.000,C 90.000,E1 123.579} C_DIS
LIN {X 0.051,Y -326.499,Z 1446.685,A 0.000,B 0.000,C 90.000,E1 123.245} C_DIS
LIN {X -0.137,Y -327.905,Z 1446.683,A 0.000,B 0.000,C 90.000,E1 122.959} C_DIS
LIN {X 0.052,Y -339.791,Z 1446.666,A 0.000,B 0.000,C 90.000,E1 119.795} C_DIS
LIN {X -0.067,Y -351.901,Z 1446.650,A 0.000,B 0.000,C 90.000,E1 117.052} C_DIS
LIN {X -0.005,Y -365.481,Z 1446.635,A 0.000,B 0.000,C 90.000,E1 114.335} C_DIS
LIN {X 0.050,Y -378.877,Z 1446.622,A 0.000,B 0.000,C 90.000,E1 111.972} C_DIS
LIN {X -0.064,Y -393.619,Z 1446.609,A 0.000,B 0.000,C 90.000,E1 109.685} C_DIS
LIN {X 0.164,Y -409.809,Z 1446.597,A 0.000,B 0.000,C 90.000,E1 107.402} C_DIS
LIN {X -0.112,Y -427.559,Z 1446.585,A 0.000,B 0.000,C 90.000,E1 105.245} C_DIS
LIN {X -0.141,Y -446.920,Z 1446.573,A 0.000,B 0.000,C 90.000,E1 103.119} C_DIS
LIN {X -0.044,Y -467.087,Z 1446.562,A 0.000,B 0.000,C 90.000,E1 101.130} C_DIS
LIN {X -0.110,Y -487.671,Z 1446.552,A 0.000,B 0.000,C 90.000,E1 99.321} C_DIS
LIN {X -0.094,Y -489.650,Z 1446.550,A 0.000,B 0.000,C 90.000,E1 99.095} C_DIS
LIN {X -0.001,Y -491.160,Z 1446.549,A 0.000,B 0.000,C 90.000,E1 98.859} C_DIS
LIN {X -0.098,Y -492.418,Z 1446.548,A 0.000,B 0.000,C 90.000,E1 98.624} C_DIS
LIN {X -0.269,Y -493.336,Z 1446.547,A 0.000,B 0.000,C 90.000,E1 98.398} C_DIS
LIN {X 0.037,Y -494.322,Z 1446.544,A 0.000,B 0.000,C 90.000,E1 97.871} C_DIS
LIN {X -0.212,Y -494.300,Z 1446.541,A 0.000,B 0.000,C 90.000,E1 97.409} C_DIS
LIN {X 0.036,Y -493.268,Z 1446.538,A 0.000,B 0.000,C 90.000,E1 96.891} C_DIS
LIN {X -0.113,Y -492.328,Z 1446.537,A 0.000,B 0.000,C 90.000,E1 96.663} C_DIS
LIN {X -0.204,Y -491.046,Z 1446.536,A 0.000,B 0.000,C 90.000,E1 96.429} C_DIS
LIN {X 0.093,Y -477.785,Z 1446.525,A 0.000,B 0.000,C 90.000,E1 94.416} C_DIS
LIN {X -0.009,Y -468.556,Z 1446.516,A 0.000,B 0.000,C 90.000,E1 92.922} C_DIS
LIN {X -0.079,Y -460.375,Z 1446.509,A 0.000,B 0.000,C 90.000,E1 91.661} C_DIS
LIN {X -0.080,Y -446.801,Z 1446.498,A 0.000,B 0.000,C 90.000,E1 89.599} C_DIS
LIN {X 0.062,Y -433.675,Z 1446.486,A 0.000,B 0.000,C 90.000,E1 87.478} C_DIS
LIN {X -0.198,Y -422.174,Z 1446.476,A 0.000,B 0.000,C 90.000,E1 85.641} C_DIS
LIN {X 0.172,Y -410.673,Z 1446.465,A 0.000,B 0.000,C 90.000,E1 83.685} C_DIS
LIN {X -0.099,Y -400.669,Z 1446.456,A 0.000,B 0.000,C 90.000,E1 82.064} C_DIS
LIN {X -0.142,Y -390.602,Z 1446.447,A 0.000,B 0.000,C 90.000,E1 80.387} C_DIS
LIN {X -0.137,Y -373.964,Z 1446.431,A 0.000,B 0.000,C 90.000,E1 77.521} C_DIS
LIN {X -0.091,Y -362.614,Z 1446.419,A 0.000,B 0.000,C 90.000,E1 75.463} C_DIS
LIN {X -0.111,Y -351.295,Z 1446.408,A 0.000,B 0.000,C 90.000,E1 73.378} C_DIS
LIN {X 0.063,Y -339.851,Z 1446.396,A 0.000,B 0.000,C 90.000,E1 71.221} C_DIS
LIN {X 0.091,Y -323.712,Z 1446.378,A 0.000,B 0.000,C 90.000,E1 68.103} C_DIS
LIN {X 0.079,Y -309.916,Z 1446.362,A 0.000,B 0.000,C 90.000,E1 65.229} C_DIS
LIN {X -0.026,Y -294.460,Z 1446.342,A 0.000,B 0.000,C 90.000,E1 61.641} C_DIS
LIN {X -0.048,Y -281.793,Z 1446.324,A 0.000,B 0.000,C 90.000,E1 58.280} C_DIS
LIN {X 0.027,Y -272.311,Z 1446.308,A 0.000,B 0.000,C 90.000,E1 55.515} C_DIS
LIN {X -0.066,Y -260.965,Z 1446.289,A 0.000,B 0.000,C 90.000,E1 52.029} C_DIS
LIN {X -0.035,Y -250.554,Z 1446.269,A 0.000,B 0.000,C 90.000,E1 48.447} C_DIS
LIN {X -0.022,Y -241.126,Z 1446.249,A 0.000,B 0.000,C 90.000,E1 44.798} C_DIS
LIN {X 0.039,Y -232.566,Z 1446.228,A 0.000,B 0.000,C 90.000,E1 41.067} C_DIS
LIN {X -0.076,Y -224.914,Z 1446.207,A 0.000,B 0.000,C 90.000,E1 37.317} C_DIS
LIN {X 0.027,Y -218.106,Z 1446.186,A 0.000,B 0.000,C 90.000,E1 33.452} C_DIS
LIN {X 0.100,Y -212.029,Z 1446.164,A 0.000,B 0.000,C 90.000,E1 29.539} C_DIS
LIN {X 0.116,Y -206.805,Z 1446.142,A 0.000,B 0.000,C 90.000,E1 25.591} C_DIS
LIN {X -0.015,Y -202.415,Z 1446.120,A 0.000,B 0.000,C 90.000,E1 21.642} C_DIS
LIN {X 0.011,Y -198.144,Z 1446.093,A 0.000,B 0.000,C 90.000,E1 16.804} C_DIS
LIN {X -0.045,Y -194.592,Z 1446.062,A 0.000,B 0.000,C 90.000,E1 11.130} C_DIS
LIN {X -0.014,Y -192.267,Z 1446.030,A 0.000,B 0.000,C 90.000,E1 5.391} C_DIS
LIN {X -0.035,Y -190.995,Z 1445.997,A 0.000,B 0.000,C 90.000,E1 359.542} C_DIS
LIN {X 0.068,Y -190.826,Z 1445.965,A 0.000,B 0.000,C 90.000,E1 353.742} C_DIS
LIN {X 0.000,Y -191.966,Z 1445.929,A 0.000,B 0.000,C 90.000,E1 347.173} C_DIS
LIN {X 0.084,Y -194.538,Z 1445.897,A 0.000,B 0.000,C 90.000,E1 341.402} C_DIS
LIN {X -0.023,Y -198.114,Z 1445.870,A 0.000,B 0.000,C 90.000,E1 336.538} C_DIS
LIN {X -0.010,Y -202.251,Z 1445.847,A 0.000,B 0.000,C 90.000,E1 332.487} C_DIS
LIN {X 0.069,Y -207.574,Z 1445.825,A 0.000,B 0.000,C 90.000,E1 328.456} C_DIS
LIN {X -0.021,Y -212.746,Z 1445.807,A 0.000,B 0.000,C 90.000,E1 325.308} C_DIS
LIN {X -0.093,Y -218.908,Z 1445.790,A 0.000,B 0.000,C 90.000,E1 322.190} C_DIS
LIN {X -0.092,Y -226.012,Z 1445.773,A 0.000,B 0.000,C 90.000,E1 319.094} C_DIS
LIN {X -0.121,Y -234.068,Z 1445.756,A 0.000,B 0.000,C 90.000,E1 316.053} C_DIS
LIN {X 0.080,Y -243.024,Z 1445.739,A 0.000,B 0.000,C 90.000,E1 313.014} C_DIS
LIN {X 0.022,Y -253.092,Z 1445.723,A 0.000,B 0.000,C 90.000,E1 310.092} C_DIS
LIN {X -0.075,Y -264.283,Z 1445.707,A 0.000,B 0.000,C 90.000,E1 307.237} C_DIS
LIN {X 0.082,Y -272.005,Z 1445.697,A 0.000,B 0.000,C 90.000,E1 305.438} C_DIS
LIN {X 0.045,Y -280.479,Z 1445.687,A 0.000,B 0.000,C 90.000,E1 303.706} C_DIS
LIN {X -0.008,Y -289.828,Z 1445.678,A 0.000,B 0.000,C 90.000,E1 302.005} C_DIS
LIN {X -0.061,Y -302.461,Z 1445.667,A 0.000,B 0.000,C 90.000,E1 300.001} C_DIS
LIN {X -0.003,Y -309.502,Z 1445.661,A 0.000,B 0.000,C 90.000,E1 298.999} C_DIS
LIN {X 0.068,Y -319.603,Z 1445.654,A 0.000,B 0.000,C 90.000,E1 297.719} C_DIS
LIN {X 0.023,Y -332.918,Z 1445.646,A 0.000,B 0.000,C 90.000,E1 296.232} C_DIS
LIN {X 0.065,Y -351.911,Z 1445.635,A 0.000,B 0.000,C 90.000,E1 294.283} C_DIS
LIN {X -0.158,Y -365.346,Z 1445.627,A 0.000,B 0.000,C 90.000,E1 292.950} C_DIS
LIN {X -0.140,Y -375.862,Z 1445.621,A 0.000,B 0.000,C 90.000,E1 291.844} C_DIS
LIN {X 0.027,Y -388.721,Z 1445.614,A 0.000,B 0.000,C 90.000,E1 290.429} C_DIS
LIN {X -0.079,Y -401.306,Z 1445.606,A 0.000,B 0.000,C 90.000,E1 289.033} C_DIS
LIN {X 0.020,Y -413.534,Z 1445.598,A 0.000,B 0.000,C 90.000,E1 287.638} C_DIS
LIN {X -0.067,Y -422.827,Z 1445.592,A 0.000,B 0.000,C 90.000,E1 286.551} C_DIS
LIN {X -0.190,Y -426.998,Z 1445.589,A 0.000,B 0.000,C 90.000,E1 286.024} C_DIS
LIN {X -0.169,Y -430.796,Z 1445.586,A 0.000,B 0.000,C 90.000,E1 285.481} C_DIS
LIN {X -0.240,Y -434.147,Z 1445.583,A 0.000,B 0.000,C 90.000,E1 284.954} C_DIS
LIN {X 0.245,Y -437.136,Z 1445.580,A 0.000,B 0.000,C 90.000,E1 284.356} C_DIS
LIN {X 0.001,Y -440.831,Z 1445.576,A 0.000,B 0.000,C 90.000,E1 283.592} C_DIS
LIN {X -0.219,Y -441.943,Z 1445.574,A 0.000,B 0.000,C 90.000,E1 283.355} C_DIS
LIN {X -0.215,Y -443.842,Z 1445.571,A 0.000,B 0.000,C 90.000,E1 282.827} C_DIS
LIN {X -0.204,Y -445.415,Z 1445.568,A 0.000,B 0.000,C 90.000,E1 282.299} C_DIS
LIN {X -0.182,Y -446.666,Z 1445.565,A 0.000,B 0.000,C 90.000,E1 281.771} C_DIS
LIN {X -0.152,Y -447.552,Z 1445.562,A 0.000,B 0.000,C 90.000,E1 281.243} C_DIS
LIN {X -0.115,Y -448.000,Z 1445.559,A 0.000,B 0.000,C 90.000,E1 280.715} C_DIS
LIN {X -0.155,Y -447.991,Z 1445.557,A 0.000,B 0.000,C 90.000,E1 280.197} C_DIS
LIN {X -0.112,Y -447.459,Z 1445.554,A 0.000,B 0.000,C 90.000,E1 279.670} C_DIS
LIN {X -0.144,Y -446.415,Z 1445.551,A 0.000,B 0.000,C 90.000,E1 279.151} C_DIS
LIN {X -0.108,Y -444.772,Z 1445.548,A 0.000,B 0.000,C 90.000,E1 278.624} C_DIS
LIN {X -0.146,Y -442.351,Z 1445.545,A 0.000,B 0.000,C 90.000,E1 278.106} C_DIS
LIN {X 0.076,Y -440.946,Z 1445.543,A 0.000,B 0.000,C 90.000,E1 277.814} C_DIS
LIN {X 0.016,Y -437.310,Z 1445.541,A 0.000,B 0.000,C 90.000,E1 277.296} C_DIS
LIN {X -0.060,Y -432.656,Z 1445.538,A 0.000,B 0.000,C 90.000,E1 276.777} C_DIS
LIN {X -0.001,Y -426.978,Z 1445.535,A 0.000,B 0.000,C 90.000,E1 276.258} C_DIS
LIN {X 0.033,Y -420.699,Z 1445.532,A 0.000,B 0.000,C 90.000,E1 275.796} C_DIS
LIN {X 0.123,Y -414.307,Z 1445.530,A 0.000,B 0.000,C 90.000,E1 275.391} C_DIS
LIN {X 0.115,Y -407.889,Z 1445.528,A 0.000,B 0.000,C 90.000,E1 275.049} C_DIS
LIN {X 0.191,Y -398.119,Z 1445.526,A 0.000,B 0.000,C 90.000,E1 274.588} C_DIS
LIN {X -0.172,Y -388.472,Z 1445.523,A 0.000,B 0.000,C 90.000,E1 274.245} C_DIS
LIN {X 0.100,Y -375.683,Z 1445.521,A 0.000,B 0.000,C 90.000,E1 273.726} C_DIS
LIN {X -0.177,Y -362.813,Z 1445.518,A 0.000,B 0.000,C 90.000,E1 273.326} C_DIS
LIN {X 0.062,Y -352.613,Z 1445.517,A 0.000,B 0.000,C 90.000,E1 272.980} C_DIS
LIN {X -0.099,Y -342.194,Z 1445.515,A 0.000,B 0.000,C 90.000,E1 272.751} C_DIS
LIN {X 0.000,Y -334.932,Z 1445.514,A 0.000,B 0.000,C 90.000,E1 272.579} C_DIS
LIN {X -0.114,Y -321.827,Z 1445.513,A 0.000,B 0.000,C 90.000,E1 272.407} C_DIS
LIN {X -0.014,Y -312.352,Z 1445.513,A 0.000,B 0.000,C 90.000,E1 272.293} C_DIS
LIN {X 0.008,Y -303.910,Z 1445.512,A 0.000,B 0.000,C 90.000,E1 272.236} C_DIS
LIN {X -0.030,Y -181.226,Z 1445.512,A 0.000,B 0.000,C 90.000,E1 272.236} C_DIS
LIN {X 0.015,Y -181.562,Z 1445.503,A 0.000,B 0.000,C 90.000,E1 270.516} C_DIS
LIN {X -0.055,Y -181.282,Z 1445.494,A 0.000,B 0.000,C 90.000,E1 268.854} C_DIS
LIN {X -0.007,Y -180.907,Z 1445.475,A 0.000,B 0.000,C 90.000,E1 265.469} C_DIS
LIN {X 0.050,Y -180.736,Z 1445.470,A 0.000,B 0.000,C 90.000,E1 264.609} C_DIS
LIN {X -0.029,Y -178.826,Z 1445.442,A 0.000,B 0.000,C 90.000,E1 259.567} C_DIS
LIN {X 0.053,Y -175.870,Z 1445.414,A 0.000,B 0.000,C 90.000,E1 254.448} C_DIS
LIN {X 0.048,Y -173.841,Z 1445.400,A 0.000,B 0.000,C 90.000,E1 251.891} C_DIS
LIN {X 0.036,Y -171.509,Z 1445.380,A 0.000,B 0.000,C 90.000,E1 248.465} C_DIS
LIN {X 0.023,Y -167.736,Z 1445.356,A 0.000,B 0.000,C 90.000,E1 244.152} C_DIS
LIN {X 0.039,Y -166.435,Z 1445.347,A 0.000,B 0.000,C 90.000,E1 242.410} C_DIS
LIN {X -0.047,Y -163.154,Z 1445.327,A 0.000,B 0.000,C 90.000,E1 238.948} C_DIS
LIN {X 0.002,Y -161.110,Z 1445.313,A 0.000,B 0.000,C 90.000,E1 236.294} C_DIS
LIN {X -0.015,Y -157.836,Z 1445.293,A 0.000,B 0.000,C 90.000,E1 232.763} C_DIS
LIN {X 0.048,Y -155.869,Z 1445.278,A 0.000,B 0.000,C 90.000,E1 230.070} C_DIS
LIN {X -0.003,Y -152.118,Z 1445.253,A 0.000,B 0.000,C 90.000,E1 225.607} C_DIS
LIN {X 0.011,Y -150.369,Z 1445.238,A 0.000,B 0.000,C 90.000,E1 222.894} C_DIS
LIN {X -0.066,Y -147.104,Z 1445.213,A 0.000,B 0.000,C 90.000,E1 218.382} C_DIS
LIN {X 0.043,Y -145.672,Z 1445.198,A 0.000,B 0.000,C 90.000,E1 215.598} C_DIS
LIN {X 0.046,Y -143.053,Z 1445.172,A 0.000,B 0.000,C 90.000,E1 211.003} C_DIS
LIN {X -0.019,Y -141.676,Z 1445.152,A 0.000,B 0.000,C 90.000,E1 207.334} C_DIS
LIN {X -0.040,Y -139.455,Z 1445.116,A 0.000,B 0.000,C 90.000,E1 200.844} C_DIS
LIN {X 0.012,Y -139.189,Z 1445.105,A 0.000,B 0.000,C 90.000,E1 198.960} C_DIS
LIN {X 0.035,Y -138.323,Z 1445.053,A 0.000,B 0.000,C 90.000,E1 189.613} C_DIS
LIN {X 0.042,Y -139.458,Z 1445.007,A 0.000,B 0.000,C 90.000,E1 181.203} C_DIS
LIN {X -0.018,Y -141.010,Z 1444.976,A 0.000,B 0.000,C 90.000,E1 175.641} C_DIS
LIN {X -0.069,Y -142.764,Z 1444.955,A 0.000,B 0.000,C 90.000,E1 171.951} C_DIS
LIN {X 0.028,Y -145.171,Z 1444.929,A 0.000,B 0.000,C 90.000,E1 167.297} C_DIS
LIN {X 0.062,Y -147.794,Z 1444.909,A 0.000,B 0.000,C 90.000,E1 163.614} C_DIS
LIN {X -0.043,Y -150.476,Z 1444.889,A 0.000,B 0.000,C 90.000,E1 160.007} C_DIS
LIN {X 0.031,Y -153.930,Z 1444.869,A 0.000,B 0.000,C 90.000,E1 156.357} C_DIS
LIN {X -0.046,Y -157.341,Z 1444.849,A 0.000,B 0.000,C 90.000,E1 152.794} C_DIS
LIN {X 0.039,Y -161.534,Z 1444.829,A 0.000,B 0.000,C 90.000,E1 149.203} C_DIS
LIN {X 0.050,Y -165.732,Z 1444.809,A 0.000,B 0.000,C 90.000,E1 145.674} C_DIS
LIN {X 0.039,Y -170.683,Z 1444.790,A 0.000,B 0.000,C 90.000,E1 142.190} C_DIS
LIN {X -0.049,Y -175.558,Z 1444.771,A 0.000,B 0.000,C 90.000,E1 138.771} C_DIS
LIN {X 0.070,Y -181.176,Z 1444.752,A 0.000,B 0.000,C 90.000,E1 135.324} C_DIS
LIN {X -0.060,Y -186.634,Z 1444.733,A 0.000,B 0.000,C 90.000,E1 132.000} C_DIS
LIN {X 0.010,Y -191.240,Z 1444.719,A 0.000,B 0.000,C 90.000,E1 129.483} C_DIS
LIN {X -0.069,Y -197.058,Z 1444.701,A 0.000,B 0.000,C 90.000,E1 126.217} C_DIS
LIN {X 0.022,Y -200.487,Z 1444.692,A 0.000,B 0.000,C 90.000,E1 124.485} C_DIS
LIN {X -0.001,Y -311.851,Z 1444.692,A 0.000,B 0.000,C 90.000,E1 124.485} C_DIS
LIN {X -0.063,Y -314.461,Z 1444.691,A 0.000,B 0.000,C 90.000,E1 124.452} C_DIS
LIN {X -0.044,Y -318.152,Z 1444.690,A 0.000,B 0.000,C 90.000,E1 124.278} C_DIS
LIN {X -0.107,Y -320.375,Z 1444.689,A 0.000,B 0.000,C 90.000,E1 124.119} C_DIS
LIN {X -0.151,Y -323.464,Z 1444.688,A 0.000,B 0.000,C 90.000,E1 123.785} C_DIS
LIN {X 0.040,Y -325.428,Z 1444.686,A 0.000,B 0.000,C 90.000,E1 123.452} C_DIS
LIN {X -0.040,Y -326.960,Z 1444.684,A 0.000,B 0.000,C 90.000,E1 123.166} C_DIS
LIN {X -0.005,Y -330.487,Z 1444.679,A 0.000,B 0.000,C 90.000,E1 122.212} C_DIS
LIN {X -0.050,Y -341.426,Z 1444.663,A 0.000,B 0.000,C 90.000,E1 119.411} C_DIS
LIN {X -0.123,Y -353.740,Z 1444.648,A 0.000,B 0.000,C 90.000,E1 116.668} C_DIS
LIN {X -0.010,Y -367.540,Z 1444.633,A 0.000,B 0.000,C 90.000,E1 113.951} C_DIS
LIN {X 0.093,Y -381.148,Z 1444.620,A 0.000,B 0.000,C 90.000,E1 111.589} C_DIS
LIN {X -0.107,Y -396.117,Z 1444.607,A 0.000,B 0.000,C 90.000,E1 109.322} C_DIS
LIN {X 0.185,Y -412.551,Z 1444.595,A 0.000,B 0.000,C 90.000,E1 107.040} C_DIS
LIN {X -0.140,Y -430.566,Z 1444.583,A 0.000,B 0.000,C 90.000,E1 104.898} C_DIS
LIN {X -0.012,Y -450.117,Z 1444.571,A 0.000,B 0.000,C 90.000,E1 102.771} C_DIS
LIN {X -0.145,Y -470.373,Z 1444.560,A 0.000,B 0.000,C 90.000,E1 100.838} C_DIS
LIN {X 0.158,Y -485.907,Z 1444.553,A 0.000,B 0.000,C 90.000,E1 99.443} C_DIS
LIN {X -0.166,Y -488.237,Z 1444.551,A 0.000,B 0.000,C 90.000,E1 99.265} C_DIS
LIN {X -0.011,Y -490.000,Z 1444.550,A 0.000,B 0.000,C 90.000,E1 99.029} C_DIS
LIN {X -0.186,Y -491.525,Z 1444.549,A 0.000,B 0.000,C 90.000,E1 98.803} C_DIS
LIN {X 0.199,Y -492.662,Z 1444.547,A 0.000,B 0.000,C 90.000,E1 98.511} C_DIS
LIN {X -0.058,Y -494.006,Z 1444.545,A 0.000,B 0.000,C 90.000,E1 98.049} C_DIS
LIN {X 0.183,Y -494.307,Z 1444.542,A 0.000,B 0.000,C 90.000,E1 97.530} C_DIS
LIN {X -0.059,Y -493.616,Z 1444.539,A 0.000,B 0.000,C 90.000,E1 97.068} C_DIS
LIN {X 0.192,Y -491.820,Z 1444.536,A 0.000,B 0.000,C 90.000,E1 96.549} C_DIS
LIN {X 0.097,Y -490.402,Z 1444.535,A 0.000,B 0.000,C 90.000,E1 96.315} C_DIS
LIN {X 0.077,Y -478.682,Z 1444.526,A 0.000,B 0.000,C 90.000,E1 94.588} C_DIS
LIN {X -0.011,Y -469.445,Z 1444.517,A 0.000,B 0.000,C 90.000,E1 93.094} C_DIS
LIN {X 0.124,Y -463.004,Z 1444.512,A 0.000,B 0.000,C 90.000,E1 92.064} C_DIS
LIN {X -0.028,Y -451.162,Z 1444.502,A 0.000,B 0.000,C 90.000,E1 90.286} C_DIS
LIN {X 0.113,Y -434.641,Z 1444.487,A 0.000,B 0.000,C 90.000,E1 87.650} C_DIS
LIN {X -0.126,Y -423.187,Z 1444.477,A 0.000,B 0.000,C 90.000,E1 85.812} C_DIS
LIN {X -0.065,Y -410.071,Z 1444.465,A 0.000,B 0.000,C 90.000,E1 83.628} C_DIS
LIN {X 0.056,Y -400.100,Z 1444.455,A 0.000,B 0.000,C 90.000,E1 81.951} C_DIS
LIN {X -0.006,Y -390.053,Z 1444.446,A 0.000,B 0.000,C 90.000,E1 80.274} C_DIS
LIN {X -0.029,Y -373.456,Z 1444.430,A 0.000,B 0.000,C 90.000,E1 77.409} C_DIS
LIN {X 0.083,Y -362.114,Z 1444.419,A 0.000,B 0.000,C 90.000,E1 75.338} C_DIS
LIN {X 0.016,Y -352.425,Z 1444.409,A 0.000,B 0.000,C 90.000,E1 73.559} C_DIS
LIN {X -0.127,Y -342.617,Z 1444.399,A 0.000,B 0.000,C 90.000,E1 71.764} C_DIS
LIN {X 0.027,Y -327.957,Z 1444.383,A 0.000,B 0.000,C 90.000,E1 68.954} C_DIS
LIN {X -0.054,Y -312.370,Z 1444.365,A 0.000,B 0.000,C 90.000,E1 65.793} C_DIS
LIN {X -0.086,Y -297.993,Z 1444.347,A 0.000,B 0.000,C 90.000,E1 62.538} C_DIS
LIN {X -0.134,Y -285.037,Z 1444.329,A 0.000,B 0.000,C 90.000,E1 59.203} C_DIS
LIN {X -0.006,Y -273.108,Z 1444.310,A 0.000,B 0.000,C 90.000,E1 55.754} C_DIS
LIN {X -0.085,Y -261.739,Z 1444.290,A 0.000,B 0.000,C 90.000,E1 52.271} C_DIS
LIN {X -0.037,Y -251.306,Z 1444.271,A 0.000,B 0.000,C 90.000,E1 48.690} C_DIS
LIN {X -0.001,Y -241.832,Z 1444.250,A 0.000,B 0.000,C 90.000,E1 45.040} C_DIS
LIN {X 0.083,Y -233.238,Z 1444.230,A 0.000,B 0.000,C 90.000,E1 41.310} C_DIS
LIN {X -0.050,Y -225.540,Z 1444.209,A 0.000,B 0.000,C 90.000,E1 37.569} C_DIS
LIN {X 0.062,Y -218.697,Z 1444.187,A 0.000,B 0.000,C 90.000,E1 33.706} C_DIS
LIN {X 0.040,Y -212.596,Z 1444.166,A 0.000,B 0.000,C 90.000,E1 29.823} C_DIS
LIN {X -0.010,Y -207.339,Z 1444.144,A 0.000,B 0.000,C 90.000,E1 25.899} C_DIS
LIN {X 0.064,Y -202.873,Z 1444.122,A 0.000,B 0.000,C 90.000,E1 21.897} C_DIS
LIN {X -0.019,Y -198.595,Z 1444.095,A 0.000,B 0.000,C 90.000,E1 17.094} C_DIS
LIN {X -0.059,Y -194.992,Z 1444.063,A 0.000,B 0.000,C 90.000,E1 11.422} C_DIS
LIN {X -0.007,Y -192.632,Z 1444.031,A 0.000,B 0.000,C 90.000,E1 5.682} C_DIS
LIN {X -0.035,Y -191.267,Z 1443.997,A 0.000,B 0.000,C 90.000,E1 359.542} C_DIS
LIN {X -0.062,Y -191.047,Z 1443.970,A 0.000,B 0.000,C 90.000,E1 354.609} C_DIS
LIN {X 0.040,Y -191.760,Z 1443.938,A 0.000,B 0.000,C 90.000,E1 348.814} C_DIS
LIN {X 0.067,Y -194.239,Z 1443.901,A 0.000,B 0.000,C 90.000,E1 342.236} C_DIS
LIN {X -0.005,Y -197.596,Z 1443.874,A 0.000,B 0.000,C 90.000,E1 337.358} C_DIS
LIN {X -0.009,Y -201.491,Z 1443.852,A 0.000,B 0.000,C 90.000,E1 333.307} C_DIS
LIN {X 0.024,Y -206.579,Z 1443.829,A 0.000,B 0.000,C 90.000,E1 329.282} C_DIS
LIN {X 0.079,Y -211.515,Z 1443.812,A 0.000,B 0.000,C 90.000,E1 326.087} C_DIS
LIN {X -0.023,Y -217.420,Z 1443.794,A 0.000,B 0.000,C 90.000,E1 322.970} C_DIS
LIN {X 0.121,Y -224.314,Z 1443.777,A 0.000,B 0.000,C 90.000,E1 319.828} C_DIS
LIN {X 0.067,Y -232.127,Z 1443.760,A 0.000,B 0.000,C 90.000,E1 316.782} C_DIS
LIN {X 0.022,Y -242.005,Z 1443.741,A 0.000,B 0.000,C 90.000,E1 313.419} C_DIS
LIN {X 0.104,Y -251.911,Z 1443.725,A 0.000,B 0.000,C 90.000,E1 310.458} C_DIS
LIN {X -0.021,Y -262.933,Z 1443.709,A 0.000,B 0.000,C 90.000,E1 307.604} C_DIS
LIN {X 0.031,Y -272.124,Z 1443.697,A 0.000,B 0.000,C 90.000,E1 305.471} C_DIS
LIN {X 0.155,Y -280.571,Z 1443.687,A 0.000,B 0.000,C 90.000,E1 303.706} C_DIS
LIN {X 0.135,Y -287.946,Z 1443.680,A 0.000,B 0.000,C 90.000,E1 302.339} C_DIS
LIN {X 0.052,Y -298.146,Z 1443.670,A 0.000,B 0.000,C 90.000,E1 300.669} C_DIS
LIN {X 0.098,Y -307.120,Z 1443.663,A 0.000,B 0.000,C 90.000,E1 299.333} C_DIS
LIN {X -0.131,Y -316.919,Z 1443.656,A 0.000,B 0.000,C 90.000,E1 298.103} C_DIS
LIN {X -0.047,Y -330.146,Z 1443.648,A 0.000,B 0.000,C 90.000,E1 296.565} C_DIS
LIN {X 0.049,Y -349.076,Z 1443.637,A 0.000,B 0.000,C 90.000,E1 294.591} C_DIS
LIN {X -0.091,Y -359.905,Z 1443.631,A 0.000,B 0.000,C 90.000,E1 293.515} C_DIS
LIN {X 0.057,Y -370.619,Z 1443.624,A 0.000,B 0.000,C 90.000,E1 292.386} C_DIS
LIN {X 0.018,Y -381.031,Z 1443.618,A 0.000,B 0.000,C 90.000,E1 291.280} C_DIS
LIN {X -0.075,Y -391.295,Z 1443.612,A 0.000,B 0.000,C 90.000,E1 290.174} C_DIS
LIN {X 0.181,Y -403.851,Z 1443.604,A 0.000,B 0.000,C 90.000,E1 288.725} C_DIS
LIN {X 0.070,Y -413.632,Z 1443.598,A 0.000,B 0.000,C 90.000,E1 287.638} C_DIS
LIN {X -0.015,Y -422.959,Z 1443.592,A 0.000,B 0.000,C 90.000,E1 286.551} C_DIS
LIN {X -0.137,Y -427.145,Z 1443.589,A 0.000,B 0.000,C 90.000,E1 286.024} C_DIS
LIN {X 0.058,Y -432.688,Z 1443.584,A 0.000,B 0.000,C 90.000,E1 285.190} C_DIS
LIN {X -0.121,Y -437.313,Z 1443.580,A 0.000,B 0.000,C 90.000,E1 284.411} C_DIS
LIN {X 0.060,Y -441.079,Z 1443.576,A 0.000,B 0.000,C 90.000,E1 283.592} C_DIS
LIN {X -0.155,Y -444.073,Z 1443.571,A 0.000,B 0.000,C 90.000,E1 282.827} C_DIS
LIN {X -0.142,Y -445.680,Z 1443.568,A 0.000,B 0.000,C 90.000,E1 282.299} C_DIS
LIN {X -0.118,Y -446.939,Z 1443.565,A 0.000,B 0.000,C 90.000,E1 281.771} C_DIS
LIN {X -0.086,Y -447.861,Z 1443.562,A 0.000,B 0.000,C 90.000,E1 281.243} C_DIS
LIN {X -0.048,Y -448.307,Z 1443.559,A 0.000,B 0.000,C 90.000,E1 280.715} C_DIS
LIN {X -0.086,Y -448.313,Z 1443.557,A 0.000,B 0.000,C 90.000,E1 280.197} C_DIS
LIN {X -0.041,Y -447.829,Z 1443.554,A 0.000,B 0.000,C 90.000,E1 279.670} C_DIS
LIN {X -0.071,Y -446.805,Z 1443.551,A 0.000,B 0.000,C 90.000,E1 279.151} C_DIS
LIN {X -0.034,Y -445.174,Z 1443.548,A 0.000,B 0.000,C 90.000,E1 278.624} C_DIS
LIN {X -0.070,Y -442.866,Z 1443.545,A 0.000,B 0.000,C 90.000,E1 278.106} C_DIS
LIN {X 0.154,Y -441.423,Z 1443.544,A 0.000,B 0.000,C 90.000,E1 277.814} C_DIS
LIN {X 0.096,Y -437.863,Z 1443.541,A 0.000,B 0.000,C 90.000,E1 277.296} C_DIS
LIN {X 0.021,Y -433.252,Z 1443.538,A 0.000,B 0.000,C 90.000,E1 276.777} C_DIS
LIN {X 0.056,Y -427.620,Z 1443.535,A 0.000,B 0.000,C 90.000,E1 276.258} C_DIS
LIN {X 0.050,Y -421.355,Z 1443.532,A 0.000,B 0.000,C 90.000,E1 275.796} C_DIS
LIN {X 0.102,Y -414.933,Z 1443.530,A 0.000,B 0.000,C 90.000,E1 275.391} C_DIS
LIN {X 0.045,Y -408.444,Z 1443.528,A 0.000,B 0.000,C 90.000,E1 275.049} C_DIS
LIN {X 0.049,Y -398.514,Z 1443.526,A 0.000,B 0.000,C 90.000,E1 274.588} C_DIS
LIN {X 0.054,Y -388.786,Z 1443.523,A 0.000,B 0.000,C 90.000,E1 274.188} C_DIS
LIN {X -0.054,Y -372.815,Z 1443.520,A 0.000,B 0.000,C 90.000,E1 273.612} C_DIS
LIN {X 0.085,Y -359.682,Z 1443.518,A 0.000,B 0.000,C 90.000,E1 273.154} C_DIS
LIN {X 0.093,Y -349.423,Z 1443.516,A 0.000,B 0.000,C 90.000,E1 272.865} C_DIS
LIN {X 0.008,Y -338.914,Z 1443.515,A 0.000,B 0.000,C 90.000,E1 272.636} C_DIS
LIN {X 0.149,Y -326.461,Z 1443.514,A 0.000,B 0.000,C 90.000,E1 272.407} C_DIS
LIN {X -0.127,Y -317.476,Z 1443.513,A 0.000,B 0.000,C 90.000,E1 272.350} C_DIS
LIN {X 0.009,Y -304.201,Z 1443.512,A 0.000,B 0.000,C 90.000,E1 272.236} C_DIS
LIN {X -0.045,Y -300.289,Z 1443.512,A 0.000,B 0.000,C 90.000,E1 272.236} C_DIS
LIN {X -0.060,Y -181.228,Z 1443.512,A 0.000,B 0.000,C 90.000,E1 272.236} C_DIS
LIN {X -0.012,Y -181.563,Z 1443.503,A 0.000,B 0.000,C 90.000,E1 270.516} C_DIS
LIN {X -0.082,Y -181.281,Z 1443.494,A 0.000,B 0.000,C 90.000,E1 268.854} C_DIS
LIN {X -0.034,Y -180.907,Z 1443.475,A 0.000,B 0.000,C 90.000,E1 265.469} C_DIS
LIN {X 0.024,Y -180.731,Z 1443.470,A 0.000,B 0.000,C 90.000,E1 264.609} C_DIS
LIN {X -0.055,Y -178.821,Z 1443.442,A 0.000,B 0.000,C 90.000,E1 259.567} C_DIS
LIN {X 0.027,Y -175.865,Z 1443.414,A 0.000,B 0.000,C 90.000,E1 254.448} C_DIS
LIN {X 0.021,Y -173.834,Z 1443.399,A 0.000,B 0.000,C 90.000,E1 251.891} C_DIS
LIN {X 0.010,Y -171.502,Z 1443.380,A 0.000,B 0.000,C 90.000,E1 248.465} C_DIS
LIN {X -0.003,Y -167.729,Z 1443.356,A 0.000,B 0.000,C 90.000,E1 244.152} C_DIS
LIN {X 0.013,Y -166.426,Z 1443.347,A 0.000,B 0.000,C 90.000,E1 242.410} C_DIS
LIN {X 0.011,Y -163.146,Z 1443.327,A 0.000,B 0.000,C 90.000,E1 238.918} C_DIS
LIN {X -0.024,Y -161.102,Z 1443.313,A 0.000,B 0.000,C 90.000,E1 236.294} C_DIS
LIN {X -0.040,Y -157.828,Z 1443.293,A 0.000,B 0.000,C 90.000,E1 232.763} C_DIS
LIN {X 0.023,Y -155.862,Z 1443.278,A 0.000,B 0.000,C 90.000,E1 230.070} C_DIS
LIN {X 0.079,Y -152.112,Z 1443.253,A 0.000,B 0.000,C 90.000,E1 225.567} C_DIS
LIN {X -0.014,Y -150.362,Z 1443.238,A 0.000,B 0.000,C 90.000,E1 222.894} C_DIS
LIN {X 0.025,Y -147.097,Z 1443.213,A 0.000,B 0.000,C 90.000,E1 218.338} C_DIS
LIN {X 0.020,Y -145.667,Z 1443.198,A 0.000,B 0.000,C 90.000,E1 215.598} C_DIS
LIN {X 0.023,Y -143.049,Z 1443.172,A 0.000,B 0.000,C 90.000,E1 211.003} C_DIS
LIN {X -0.042,Y -141.672,Z 1443.152,A 0.000,B 0.000,C 90.000,E1 207.334} C_DIS
LIN {X 0.068,Y -139.453,Z 1443.116,A 0.000,B 0.000,C 90.000,E1 200.791} C_DIS
LIN {X -0.011,Y -139.187,Z 1443.105,A 0.000,B 0.000,C 90.000,E1 198.960} C_DIS
LIN {X 0.011,Y -138.322,Z 1443.053,A 0.000,B 0.000,C 90.000,E1 189.613} C_DIS
LIN {X 0.019,Y -139.459,Z 1443.007,A 0.000,B 0.000,C 90.000,E1 181.203} C_DIS
LIN {X -0.041,Y -141.014,Z 1442.976,A 0.000,B 0.000,C 90.000,E1 175.641} C_DIS
LIN {X 0.049,Y -142.767,Z 1442.955,A 0.000,B 0.000,C 90.000,E1 171.894} C_DIS
LIN {X 0.005,Y -145.177,Z 1442.929,A 0.000,B 0.000,C 90.000,E1 167.297} C_DIS
LIN {X 0.038,Y -147.800,Z 1442.909,A 0.000,B 0.000,C 90.000,E1 163.614} C_DIS
LIN {X -0.067,Y -150.484,Z 1442.889,A 0.000,B 0.000,C 90.000,E1 160.007} C_DIS
LIN {X 0.007,Y -153.939,Z 1442.869,A 0.000,B 0.000,C 90.000,E1 156.357} C_DIS
LIN {X 0.069,Y -157.350,Z 1442.849,A 0.000,B 0.000,C 90.000,E1 152.743} C_DIS
LIN {X 0.013,Y -161.546,Z 1442.829,A 0.000,B 0.000,C 90.000,E1 149.203} C_DIS
LIN {X 0.025,Y -165.744,Z 1442.809,A 0.000,B 0.000,C 90.000,E1 145.674} C_DIS
LIN {X 0.013,Y -170.697,Z 1442.790,A 0.000,B 0.000,C 90.000,E1 142.190} C_DIS
LIN {X -0.076,Y -175.571,Z 1442.771,A 0.000,B 0.000,C 90.000,E1 138.771} C_DIS
LIN {X 0.043,Y -181.189,Z 1442.752,A 0.000,B 0.000,C 90.000,E1 135.324} C_DIS
LIN {X -0.088,Y -186.649,Z 1442.733,A 0.000,B 0.000,C 90.000,E1 132.000} C_DIS
LIN {X -0.019,Y -191.254,Z 1442.719,A 0.000,B 0.000,C 90.000,E1 129.483} C_DIS
LIN {X 0.062,Y -197.074,Z 1442.701,A 0.000,B 0.000,C 90.000,E1 126.171} C_DIS
LIN {X -0.059,Y -200.439,Z 1442.692,A 0.000,B 0.000,C 90.000,E1 124.532} C_DIS
LIN {X 0.113,Y -312.301,Z 1442.692,A 0.000,B 0.000,C 90.000,E1 124.485} C_DIS
LIN {X -0.088,Y -317.817,Z 1442.691,A 0.000,B 0.000,C 90.000,E1 124.326} C_DIS
LIN {X 0.023,Y -320.283,Z 1442.690,A 0.000,B 0.000,C 90.000,E1 124.119} C_DIS
LIN {X -0.197,Y -323.599,Z 1442.688,A 0.000,B 0.000,C 90.000,E1 123.785} C_DIS
LIN {X -0.029,Y -325.528,Z 1442.686,A 0.000,B 0.000,C 90.000,E1 123.452} C_DIS
LIN {X -0.131,Y -327.035,Z 1442.684,A 0.000,B 0.000,C 90.000,E1 123.166} C_DIS
LIN {X -0.143,Y -341.470,Z 1442.663,A 0.000,B 0.000,C 90.000,E1 119.411} C_DIS
LIN {X 0.097,Y -353.791,Z 1442.648,A 0.000,B 0.000,C 90.000,E1 116.616} C_DIS
LIN {X -0.108,Y -367.600,Z 1442.633,A 0.000,B 0.000,C 90.000,E1 113.951} C_DIS
LIN {X -0.007,Y -381.216,Z 1442.620,A 0.000,B 0.000,C 90.000,E1 111.589} C_DIS
LIN {X 0.165,Y -396.194,Z 1442.607,A 0.000,B 0.000,C 90.000,E1 109.268} C_DIS
LIN {X 0.081,Y -412.638,Z 1442.595,A 0.000,B 0.000,C 90.000,E1 107.040} C_DIS
LIN {X -0.136,Y -430.663,Z 1442.583,A 0.000,B 0.000,C 90.000,E1 104.883} C_DIS
LIN {X -0.119,Y -450.222,Z 1442.571,A 0.000,B 0.000,C 90.000,E1 102.771} C_DIS
LIN {X -0.249,Y -470.482,Z 1442.560,A 0.000,B 0.000,C 90.000,E1 100.838} C_DIS
LIN {X 0.058,Y -486.018,Z 1442.552,A 0.000,B 0.000,C 90.000,E1 99.443} C_DIS
LIN {X 0.216,Y -488.294,Z 1442.551,A 0.000,B 0.000,C 90.000,E1 99.208} C_DIS
LIN {X -0.110,Y -490.016,Z 1442.550,A 0.000,B 0.000,C 90.000,E1 99.029} C_DIS
LIN {X 0.199,Y -491.508,Z 1442.549,A 0.000,B 0.000,C 90.000,E1 98.746} C_DIS
LIN {X 0.100,Y -492.618,Z 1442.547,A 0.000,B 0.000,C 90.000,E1 98.511} C_DIS
LIN {X -0.158,Y -493.921,Z 1442.545,A 0.000,B 0.000,C 90.000,E1 98.049} C_DIS
LIN {X 0.082,Y -494.185,Z 1442.542,A 0.000,B 0.000,C 90.000,E1 97.530} C_DIS
LIN {X -0.160,Y -493.456,Z 1442.539,A 0.000,B 0.000,C 90.000,E1 97.068} C_DIS
LIN {X 0.090,Y -491.616,Z 1442.536,A 0.000,B 0.000,C 90.000,E1 96.549} C_DIS
LIN {X -0.005,Y -490.167,Z 1442.535,A 0.000,B 0.000,C 90.000,E1 96.315} C_DIS
LIN {X -0.027,Y -478.454,Z 1442.526,A 0.000,B 0.000,C 90.000,E1 94.588} C_DIS
LIN {X -0.117,Y -469.191,Z 1442.517,A 0.000,B 0.000,C 90.000,E1 93.094} C_DIS
LIN {X -0.177,Y -461.057,Z 1442.510,A 0.000,B 0.000,C 90.000,E1 91.833} C_DIS
LIN {X -0.161,Y -447.516,Z 1442.499,A 0.000,B 0.000,C 90.000,E1 89.771} C_DIS
LIN {X 0.161,Y -432.794,Z 1442.485,A 0.000,B 0.000,C 90.000,E1 87.364} C_DIS
LIN {X -0.125,Y -421.348,Z 1442.475,A 0.000,B 0.000,C 90.000,E1 85.527} C_DIS
LIN {X -0.180,Y -409.915,Z 1442.464,A 0.000,B 0.000,C 90.000,E1 83.628} C_DIS
LIN {X -0.059,Y -399.986,Z 1442.455,A 0.000,B 0.000,C 90.000,E1 81.951} C_DIS
LIN {X -0.119,Y -389.948,Z 1442.446,A 0.000,B 0.000,C 90.000,E1 80.274} C_DIS
LIN {X -0.141,Y -373.374,Z 1442.430,A 0.000,B 0.000,C 90.000,E1 77.409} C_DIS
LIN {X -0.027,Y -362.049,Z 1442.419,A 0.000,B 0.000,C 90.000,E1 75.338} C_DIS
LIN {X -0.091,Y -352.351,Z 1442.409,A 0.000,B 0.000,C 90.000,E1 73.559} C_DIS
LIN {X 0.091,Y -342.542,Z 1442.398,A 0.000,B 0.000,C 90.000,E1 71.710} C_DIS
LIN {X -0.077,Y -327.844,Z 1442.383,A 0.000,B 0.000,C 90.000,E1 68.954} C_DIS
LIN {X -0.088,Y -313.742,Z 1442.367,A 0.000,B 0.000,C 90.000,E1 66.102} C_DIS
LIN {X -0.093,Y -300.632,Z 1442.351,A 0.000,B 0.000,C 90.000,E1 63.179} C_DIS
LIN {X 0.029,Y -286.173,Z 1442.331,A 0.000,B 0.000,C 90.000,E1 59.488} C_DIS
LIN {X -0.048,Y -274.194,Z 1442.312,A 0.000,B 0.000,C 90.000,E1 56.087} C_DIS
LIN {X 0.062,Y -263.924,Z 1442.294,A 0.000,B 0.000,C 90.000,E1 52.924} C_DIS
LIN {X 0.000,Y -253.332,Z 1442.274,A 0.000,B 0.000,C 90.000,E1 49.380} C_DIS
LIN {X 0.100,Y -243.709,Z 1442.254,A 0.000,B 0.000,C 90.000,E1 45.729} C_DIS
LIN {X -0.099,Y -234.970,Z 1442.234,A 0.000,B 0.000,C 90.000,E1 42.081} C_DIS
LIN {X -0.025,Y -227.097,Z 1442.213,A 0.000,B 0.000,C 90.000,E1 38.302} C_DIS
LIN {X -0.042,Y -220.113,Z 1442.192,A 0.000,B 0.000,C 90.000,E1 34.485} C_DIS
LIN {X 0.026,Y -213.913,Z 1442.170,A 0.000,B 0.000,C 90.000,E1 30.590} C_DIS
LIN {X 0.010,Y -208.503,Z 1442.148,A 0.000,B 0.000,C 90.000,E1 26.668} C_DIS
LIN {X 0.015,Y -203.875,Z 1442.126,A 0.000,B 0.000,C 90.000,E1 22.695} C_DIS
LIN {X 0.032,Y -199.465,Z 1442.099,A 0.000,B 0.000,C 90.000,E1 17.873} C_DIS
LIN {X 0.075,Y -195.678,Z 1442.068,A 0.000,B 0.000,C 90.000,E1 12.187} C_DIS
LIN {X 0.021,Y -193.153,Z 1442.036,A 0.000,B 0.000,C 90.000,E1 6.486} C_DIS
LIN {X 0.006,Y -191.707,Z 1442.004,A 0.000,B 0.000,C 90.000,E1 0.745} C_DIS
LIN {X 0.077,Y -191.323,Z 1441.979,A 0.000,B 0.000,C 90.000,E1 356.216} C_DIS
LIN {X -0.018,Y -191.470,Z 1441.956,A 0.000,B 0.000,C 90.000,E1 352.129} C_DIS
LIN {X 0.087,Y -192.937,Z 1441.920,A 0.000,B 0.000,C 90.000,E1 345.519} C_DIS
LIN {X -0.045,Y -195.950,Z 1441.888,A 0.000,B 0.000,C 90.000,E1 339.826} C_DIS
LIN {X 0.046,Y -199.960,Z 1441.861,A 0.000,B 0.000,C 90.000,E1 334.921} C_DIS
LIN {X -0.068,Y -204.600,Z 1441.838,A 0.000,B 0.000,C 90.000,E1 330.923} C_DIS
LIN {X 0.010,Y -210.365,Z 1441.816,A 0.000,B 0.000,C 90.000,E1 326.914} C_DIS
LIN {X -0.074,Y -216.004,Z 1441.799,A 0.000,B 0.000,C 90.000,E1 323.783} C_DIS
LIN {X 0.026,Y -222.667,Z 1441.781,A 0.000,B 0.000,C 90.000,E1 320.642} C_DIS
LIN {X 0.102,Y -230.244,Z 1441.764,A 0.000,B 0.000,C 90.000,E1 317.553} C_DIS
LIN {X 0.002,Y -239.852,Z 1441.745,A 0.000,B 0.000,C 90.000,E1 314.190} C_DIS
LIN {X 0.026,Y -249.492,Z 1441.729,A 0.000,B 0.000,C 90.000,E1 311.229} C_DIS
LIN {X 0.000,Y -260.185,Z 1441.713,A 0.000,B 0.000,C 90.000,E1 308.338} C_DIS
LIN {X 0.007,Y -270.624,Z 1441.699,A 0.000,B 0.000,C 90.000,E1 305.851} C_DIS
LIN {X -0.114,Y -280.664,Z 1441.688,A 0.000,B 0.000,C 90.000,E1 303.785} C_DIS
LIN {X -0.138,Y -288.018,Z 1441.680,A 0.000,B 0.000,C 90.000,E1 302.418} C_DIS
LIN {X -0.075,Y -298.179,Z 1441.671,A 0.000,B 0.000,C 90.000,E1 300.718} C_DIS
LIN {X -0.186,Y -307.149,Z 1441.663,A 0.000,B 0.000,C 90.000,E1 299.411} C_DIS
LIN {X 0.078,Y -316.834,Z 1441.656,A 0.000,B 0.000,C 90.000,E1 298.103} C_DIS
LIN {X -0.148,Y -330.046,Z 1441.648,A 0.000,B 0.000,C 90.000,E1 296.616} C_DIS
LIN {X -0.111,Y -349.034,Z 1441.637,A 0.000,B 0.000,C 90.000,E1 294.643} C_DIS
LIN {X -0.035,Y -359.495,Z 1441.631,A 0.000,B 0.000,C 90.000,E1 293.567} C_DIS
LIN {X -0.034,Y -370.198,Z 1441.625,A 0.000,B 0.000,C 90.000,E1 292.461} C_DIS
LIN {X -0.065,Y -380.609,Z 1441.619,A 0.000,B 0.000,C 90.000,E1 291.354} C_DIS
LIN {X -0.154,Y -390.852,Z 1441.612,A 0.000,B 0.000,C 90.000,E1 290.248} C_DIS
LIN {X -0.132,Y -403.404,Z 1441.604,A 0.000,B 0.000,C 90.000,E1 288.833} C_DIS
LIN {X 0.165,Y -415.693,Z 1441.597,A 0.000,B 0.000,C 90.000,E1 287.402} C_DIS
LIN {X -0.153,Y -422.700,Z 1441.592,A 0.000,B 0.000,C 90.000,E1 286.622} C_DIS
LIN {X -0.158,Y -426.948,Z 1441.589,A 0.000,B 0.000,C 90.000,E1 286.079} C_DIS
LIN {X -0.138,Y -430.793,Z 1441.586,A 0.000,B 0.000,C 90.000,E1 285.536} C_DIS
LIN {X -0.024,Y -435.779,Z 1441.582,A 0.000,B 0.000,C 90.000,E1 284.717} C_DIS
LIN {X 0.048,Y -438.616,Z 1441.579,A 0.000,B 0.000,C 90.000,E1 284.175} C_DIS
LIN {X -0.190,Y -442.162,Z 1441.574,A 0.000,B 0.000,C 90.000,E1 283.411} C_DIS
LIN {X -0.186,Y -444.138,Z 1441.571,A 0.000,B 0.000,C 90.000,E1 282.883} C_DIS
LIN {X -0.174,Y -445.802,Z 1441.568,A 0.000,B 0.000,C 90.000,E1 282.355} C_DIS
LIN {X -0.151,Y -447.142,Z 1441.566,A 0.000,B 0.000,C 90.000,E1 281.827} C_DIS
LIN {X -0.120,Y -448.048,Z 1441.563,A 0.000,B 0.000,C 90.000,E1 281.299} C_DIS
LIN {X -0.164,Y -448.577,Z 1441.560,A 0.000,B 0.000,C 90.000,E1 280.782} C_DIS
LIN {X -0.119,Y -448.660,Z 1441.557,A 0.000,B 0.000,C 90.000,E1 280.254} C_DIS
LIN {X -0.073,Y -448.237,Z 1441.554,A 0.000,B 0.000,C 90.000,E1 279.726} C_DIS
LIN {X -0.102,Y -447.283,Z 1441.551,A 0.000,B 0.000,C 90.000,E1 279.208} C_DIS
LIN {X -0.063,Y -445.734,Z 1441.548,A 0.000,B 0.000,C 90.000,E1 278.681} C_DIS
LIN {X -0.096,Y -443.516,Z 1441.545,A 0.000,B 0.000,C 90.000,E1 278.163} C_DIS
LIN {X 0.130,Y -442.146,Z 1441.544,A 0.000,B 0.000,C 90.000,E1 277.871} C_DIS
LIN {X 0.075,Y -438.690,Z 1441.541,A 0.000,B 0.000,C 90.000,E1 277.352} C_DIS
LIN {X -0.200,Y -436.629,Z 1441.539,A 0.000,B 0.000,C 90.000,E1 277.125} C_DIS
LIN {X 0.155,Y -431.618,Z 1441.536,A 0.000,B 0.000,C 90.000,E1 276.549} C_DIS
LIN {X -0.009,Y -428.768,Z 1441.535,A 0.000,B 0.000,C 90.000,E1 276.315} C_DIS
LIN {X -0.099,Y -422.522,Z 1441.532,A 0.000,B 0.000,C 90.000,E1 275.853} C_DIS
LIN {X -0.115,Y -416.130,Z 1441.530,A 0.000,B 0.000,C 90.000,E1 275.448} C_DIS
LIN {X -0.179,Y -406.271,Z 1441.527,A 0.000,B 0.000,C 90.000,E1 274.935} C_DIS
LIN {X 0.009,Y -396.509,Z 1441.525,A 0.000,B 0.000,C 90.000,E1 274.473} C_DIS
LIN {X 0.052,Y -386.714,Z 1441.523,A 0.000,B 0.000,C 90.000,E1 274.073} C_DIS
LIN {X -0.022,Y -373.931,Z 1441.520,A 0.000,B 0.000,C 90.000,E1 273.612} C_DIS
LIN {X 0.119,Y -360.792,Z 1441.518,A 0.000,B 0.000,C 90.000,E1 273.154} C_DIS
LIN {X 0.117,Y -350.516,Z 1441.516,A 0.000,B 0.000,C 90.000,E1 272.865} C_DIS
LIN {X 0.001,Y -339.720,Z 1441.515,A 0.000,B 0.000,C 90.000,E1 272.636} C_DIS
LIN {X -0.148,Y -327.923,Z 1441.514,A 0.000,B 0.000,C 90.000,E1 272.465} C_DIS
LIN {X -0.103,Y -318.827,Z 1441.513,A 0.000,B 0.000,C 90.000,E1 272.350} C_DIS
LIN {X 0.031,Y -305.666,Z 1441.512,A 0.000,B 0.000,C 90.000,E1 272.236} C_DIS
LIN {X -0.023,Y -303.112,Z 1441.512,A 0.000,B 0.000,C 90.000,E1 272.236} C_DIS
LIN {X -0.047,Y -181.227,Z 1441.512,A 0.000,B 0.000,C 90.000,E1 272.236} C_DIS
LIN {X 0.000,Y -181.562,Z 1441.503,A 0.000,B 0.000,C 90.000,E1 270.516} C_DIS
LIN {X -0.070,Y -181.282,Z 1441.494,A 0.000,B 0.000,C 90.000,E1 268.854} C_DIS
LIN {X -0.021,Y -180.907,Z 1441.475,A 0.000,B 0.000,C 90.000,E1 265.469} C_DIS
LIN {X 0.036,Y -180.733,Z 1441.470,A 0.000,B 0.000,C 90.000,E1 264.609} C_DIS
LIN {X -0.043,Y -178.823,Z 1441.442,A 0.000,B 0.000,C 90.000,E1 259.567} C_DIS
LIN {X 0.039,Y -175.867,Z 1441.414,A 0.000,B 0.000,C 90.000,E1 254.448} C_DIS
LIN {X 0.033,Y -173.838,Z 1441.399,A 0.000,B 0.000,C 90.000,E1 251.891} C_DIS
LIN {X 0.022,Y -171.506,Z 1441.380,A 0.000,B 0.000,C 90.000,E1 248.465} C_DIS
LIN {X 0.009,Y -167.733,Z 1441.356,A 0.000,B 0.000,C 90.000,E1 244.152} C_DIS
LIN {X 0.025,Y -166.429,Z 1441.347,A 0.000,B 0.000,C 90.000,E1 242.410} C_DIS
LIN {X -0.061,Y -163.149,Z 1441.327,A 0.000,B 0.000,C 90.000,E1 238.948} C_DIS
LIN {X -0.012,Y -161.105,Z 1441.313,A 0.000,B 0.000,C 90.000,E1 236.294} C_DIS
LIN {X -0.028,Y -157.832,Z 1441.293,A 0.000,B 0.000,C 90.000,E1 232.763} C_DIS
LIN {X 0.035,Y -155.865,Z 1441.278,A 0.000,B 0.000,C 90.000,E1 230.070} C_DIS
LIN {X 0.090,Y -152.115,Z 1441.253,A 0.000,B 0.000,C 90.000,E1 225.567} C_DIS
LIN {X -0.001,Y -150.365,Z 1441.238,A 0.000,B 0.000,C 90.000,E1 222.894} C_DIS
LIN {X 0.037,Y -147.100,Z 1441.213,A 0.000,B 0.000,C 90.000,E1 218.338} C_DIS
LIN {X 0.031,Y -145.669,Z 1441.198,A 0.000,B 0.000,C 90.000,E1 215.598} C_DIS
LIN {X 0.034,Y -143.051,Z 1441.172,A 0.000,B 0.000,C 90.000,E1 211.003} C_DIS
LIN {X -0.031,Y -141.674,Z 1441.152,A 0.000,B 0.000,C 90.000,E1 207.334} C_DIS
LIN {X 0.078,Y -139.454,Z 1441.116,A 0.000,B 0.000,C 90.000,E1 200.791} C_DIS
LIN {X -0.001,Y -139.187,Z 1441.105,A 0.000,B 0.000,C 90.000,E1 198.960} C_DIS
LIN {X 0.022,Y -138.323,Z 1441.053,A 0.000,B 0.000,C 90.000,E1 189.613} C_DIS
LIN {X 0.029,Y -139.458,Z 1441.007,A 0.000,B 0.000,C 90.000,E1 181.203} C_DIS
LIN {X -0.030,Y -141.012,Z 1440.976,A 0.000,B 0.000,C 90.000,E1 175.641} C_DIS
LIN {X 0.060,Y -142.766,Z 1440.955,A 0.000,B 0.000,C 90.000,E1 171.894} C_DIS
LIN {X 0.015,Y -145.175,Z 1440.929,A 0.000,B 0.000,C 90.000,E1 167.297} C_DIS
LIN {X 0.049,Y -147.796,Z 1440.909,A 0.000,B 0.000,C 90.000,E1 163.614} C_DIS
LIN {X -0.055,Y -150.481,Z 1440.889,A 0.000,B 0.000,C 90.000,E1 160.007} C_DIS
LIN {X 0.018,Y -153.935,Z 1440.869,A 0.000,B 0.000,C 90.000,E1 156.357} C_DIS
LIN {X 0.081,Y -157.346,Z 1440.849,A 0.000,B 0.000,C 90.000,E1 152.743} C_DIS
LIN {X 0.024,Y -161.541,Z 1440.829,A 0.000,B 0.000,C 90.000,E1 149.203} C_DIS
LIN {X 0.037,Y -165.739,Z 1440.809,A 0.000,B 0.000,C 90.000,E1 145.674} C_DIS
LIN {X 0.025,Y -170.691,Z 1440.790,A 0.000,B 0.000,C 90.000,E1 142.190} C_DIS
LIN {X -0.064,Y -175.565,Z 1440.771,A 0.000,B 0.000,C 90.000,E1 138.771} C_DIS
LIN {X 0.056,Y -181.183,Z 1440.752,A 0.000,B 0.000,C 90.000,E1 135.324} C_DIS
LIN {X -0.075,Y -186.642,Z 1440.733,A 0.000,B 0.000,C 90.000,E1 132.000} C_DIS
LIN {X -0.006,Y -191.248,Z 1440.719,A 0.000,B 0.000,C 90.000,E1 129.483} C_DIS
LIN {X 0.075,Y -197.067,Z 1440.701,A 0.000,B 0.000,C 90.000,E1 126.171} C_DIS
LIN {X 0.021,Y -200.394,Z 1440.692,A 0.000,B 0.000,C 90.000,E1 124.532} C_DIS
LIN {X -0.019,Y -312.334,Z 1440.692,A 0.000,B 0.000,C 90.000,E1 124.532} C_DIS
LIN {X 0.082,Y -313.905,Z 1440.692,A 0.000,B 0.000,C 90.000,E1 124.485} C_DIS
LIN {X -0.067,Y -318.041,Z 1440.691,A 0.000,B 0.000,C 90.000,E1 124.326} C_DIS
LIN {X 0.045,Y -320.409,Z 1440.690,A 0.000,B 0.000,C 90.000,E1 124.119} C_DIS
LIN {X -0.176,Y -323.644,Z 1440.688,A 0.000,B 0.000,C 90.000,E1 123.785} C_DIS
LIN {X -0.037,Y -325.567,Z 1440.686,A 0.000,B 0.000,C 90.000,E1 123.452} C_DIS
LIN {X -0.171,Y -327.065,Z 1440.684,A 0.000,B 0.000,C 90.000,E1 123.166} C_DIS
LIN {X -0.184,Y -341.477,Z 1440.663,A 0.000,B 0.000,C 90.000,E1 119.411} C_DIS
LIN {X 0.055,Y -353.801,Z 1440.648,A 0.000,B 0.000,C 90.000,E1 116.616} C_DIS
LIN {X -0.152,Y -367.614,Z 1440.633,A 0.000,B 0.000,C 90.000,E1 113.951} C_DIS
LIN {X -0.053,Y -381.233,Z 1440.620,A 0.000,B 0.000,C 90.000,E1 111.589} C_DIS
LIN {X 0.118,Y -396.216,Z 1440.607,A 0.000,B 0.000,C 90.000,E1 109.268} C_DIS
LIN {X 0.032,Y -412.663,Z 1440.595,A 0.000,B 0.000,C 90.000,E1 107.040} C_DIS
LIN {X 0.231,Y -430.693,Z 1440.583,A 0.000,B 0.000,C 90.000,E1 104.828} C_DIS
LIN {X -0.168,Y -450.256,Z 1440.571,A 0.000,B 0.000,C 90.000,E1 102.771} C_DIS
LIN {X 0.165,Y -470.517,Z 1440.560,A 0.000,B 0.000,C 90.000,E1 100.782} C_DIS
LIN {X 0.010,Y -486.055,Z 1440.552,A 0.000,B 0.000,C 90.000,E1 99.443} C_DIS
LIN {X 0.168,Y -488.292,Z 1440.551,A 0.000,B 0.000,C 90.000,E1 99.208} C_DIS
LIN {X -0.157,Y -489.986,Z 1440.550,A 0.000,B 0.000,C 90.000,E1 99.029} C_DIS
LIN {X 0.151,Y -491.456,Z 1440.549,A 0.000,B 0.000,C 90.000,E1 98.746} C_DIS
LIN {X 0.051,Y -492.548,Z 1440.547,A 0.000,B 0.000,C 90.000,E1 98.511} C_DIS
LIN {X -0.206,Y -493.822,Z 1440.545,A 0.000,B 0.000,C 90.000,E1 98.049} C_DIS
LIN {X 0.033,Y -494.061,Z 1440.542,A 0.000,B 0.000,C 90.000,E1 97.530} C_DIS
LIN {X -0.209,Y -493.307,Z 1440.539,A 0.000,B 0.000,C 90.000,E1 97.068} C_DIS
LIN {X 0.040,Y -491.434,Z 1440.536,A 0.000,B 0.000,C 90.000,E1 96.549} C_DIS
LIN {X -0.203,Y -488.255,Z 1440.534,A 0.000,B 0.000,C 90.000,E1 96.087} C_DIS
LIN {X -0.079,Y -478.269,Z 1440.525,A 0.000,B 0.000,C 90.000,E1 94.588} C_DIS
LIN {X -0.172,Y -468.983,Z 1440.517,A 0.000,B 0.000,C 90.000,E1 93.094} C_DIS
LIN {X 0.226,Y -460.828,Z 1440.510,A 0.000,B 0.000,C 90.000,E1 91.776} C_DIS
LIN {X -0.221,Y -447.298,Z 1440.499,A 0.000,B 0.000,C 90.000,E1 89.771} C_DIS
LIN {X 0.097,Y -432.614,Z 1440.485,A 0.000,B 0.000,C 90.000,E1 87.364} C_DIS
LIN {X -0.190,Y -421.203,Z 1440.475,A 0.000,B 0.000,C 90.000,E1 85.527} C_DIS
LIN {X 0.161,Y -409.784,Z 1440.464,A 0.000,B 0.000,C 90.000,E1 83.571} C_DIS
LIN {X -0.041,Y -398.237,Z 1440.454,A 0.000,B 0.000,C 90.000,E1 81.659} C_DIS
LIN {X -0.131,Y -388.207,Z 1440.444,A 0.000,B 0.000,C 90.000,E1 79.982} C_DIS
LIN {X -0.203,Y -371.696,Z 1440.428,A 0.000,B 0.000,C 90.000,E1 77.117} C_DIS
LIN {X -0.119,Y -360.400,Z 1440.417,A 0.000,B 0.000,C 90.000,E1 75.046} C_DIS
LIN {X -0.114,Y -350.692,Z 1440.407,A 0.000,B 0.000,C 90.000,E1 73.251} C_DIS
LIN {X 0.042,Y -340.818,Z 1440.397,A 0.000,B 0.000,C 90.000,E1 71.402} C_DIS
LIN {X 0.167,Y -327.775,Z 1440.383,A 0.000,B 0.000,C 90.000,E1 68.901} C_DIS
LIN {X 0.138,Y -313.650,Z 1440.367,A 0.000,B 0.000,C 90.000,E1 66.049} C_DIS
LIN {X 0.088,Y -301.933,Z 1440.353,A 0.000,B 0.000,C 90.000,E1 63.461} C_DIS
LIN {X 0.143,Y -288.599,Z 1440.334,A 0.000,B 0.000,C 90.000,E1 60.127} C_DIS
LIN {X -0.004,Y -276.477,Z 1440.315,A 0.000,B 0.000,C 90.000,E1 56.755} C_DIS
LIN {X 0.022,Y -266.181,Z 1440.298,A 0.000,B 0.000,C 90.000,E1 53.623} C_DIS
LIN {X 0.065,Y -255.391,Z 1440.278,A 0.000,B 0.000,C 90.000,E1 50.070} C_DIS
LIN {X 0.056,Y -245.639,Z 1440.258,A 0.000,B 0.000,C 90.000,E1 46.458} C_DIS
LIN {X 0.076,Y -236.729,Z 1440.238,A 0.000,B 0.000,C 90.000,E1 42.771} C_DIS
LIN {X 0.025,Y -228.715,Z 1440.217,A 0.000,B 0.000,C 90.000,E1 39.036} C_DIS
LIN {X 0.005,Y -221.564,Z 1440.196,A 0.000,B 0.000,C 90.000,E1 35.231} C_DIS
LIN {X -0.070,Y -215.242,Z 1440.174,A 0.000,B 0.000,C 90.000,E1 31.386} C_DIS
LIN {X -0.039,Y -209.662,Z 1440.152,A 0.000,B 0.000,C 90.000,E1 27.462} C_DIS
LIN {X -0.088,Y -204.928,Z 1440.130,A 0.000,B 0.000,C 90.000,E1 23.515} C_DIS
LIN {X 0.048,Y -200.352,Z 1440.104,A 0.000,B 0.000,C 90.000,E1 18.671} C_DIS
LIN {X 0.017,Y -196.864,Z 1440.077,A 0.000,B 0.000,C 90.000,E1 13.828} C_DIS
LIN {X -0.087,Y -194.356,Z 1440.050,A 0.000,B 0.000,C 90.000,E1 8.973} C_DIS
LIN {X 0.080,Y -192.664,Z 1440.022,A 0.000,B 0.000,C 90.000,E1 4.012} C_DIS
LIN {X 0.089,Y -191.754,Z 1439.993,A 0.000,B 0.000,C 90.000,E1 358.682} C_DIS
LIN {X -0.085,Y -191.634,Z 1439.965,A 0.000,B 0.000,C 90.000,E1 353.799} C_DIS
LIN {X 0.080,Y -192.400,Z 1439.933,A 0.000,B 0.000,C 90.000,E1 347.993} C_DIS
LIN {X 0.003,Y -195.093,Z 1439.897,A 0.000,B 0.000,C 90.000,E1 341.456} C_DIS
LIN {X 0.025,Y -198.673,Z 1439.870,A 0.000,B 0.000,C 90.000,E1 336.561} C_DIS
LIN {X -0.042,Y -202.816,Z 1439.847,A 0.000,B 0.000,C 90.000,E1 332.538} C_DIS
LIN {X -0.049,Y -208.076,Z 1439.825,A 0.000,B 0.000,C 90.000,E1 328.535} C_DIS
LIN {X 0.043,Y -213.208,Z 1439.807,A 0.000,B 0.000,C 90.000,E1 325.341} C_DIS
LIN {X 0.109,Y -219.358,Z 1439.790,A 0.000,B 0.000,C 90.000,E1 322.190} C_DIS
LIN {X -0.043,Y -226.492,Z 1439.773,A 0.000,B 0.000,C 90.000,E1 319.138} C_DIS
LIN {X -0.087,Y -235.624,Z 1439.754,A 0.000,B 0.000,C 90.000,E1 315.729} C_DIS
LIN {X -0.022,Y -244.699,Z 1439.737,A 0.000,B 0.000,C 90.000,E1 312.732} C_DIS
LIN {X 0.000,Y -256.174,Z 1439.719,A 0.000,B 0.000,C 90.000,E1 309.439} C_DIS
LIN {X -0.073,Y -266.120,Z 1439.705,A 0.000,B 0.000,C 90.000,E1 306.950} C_DIS
LIN {X 0.037,Y -275.638,Z 1439.693,A 0.000,B 0.000,C 90.000,E1 304.818} C_DIS
LIN {X 0.019,Y -286.166,Z 1439.682,A 0.000,B 0.000,C 90.000,E1 302.752} C_DIS
LIN {X 0.052,Y -296.125,Z 1439.673,A 0.000,B 0.000,C 90.000,E1 301.052} C_DIS
LIN {X -0.082,Y -304.865,Z 1439.665,A 0.000,B 0.000,C 90.000,E1 299.745} C_DIS
LIN {X 0.087,Y -311.936,Z 1439.660,A 0.000,B 0.000,C 90.000,E1 298.743} C_DIS
LIN {X -0.164,Y -324.575,Z 1439.651,A 0.000,B 0.000,C 90.000,E1 297.257} C_DIS
LIN {X 0.089,Y -340.843,Z 1439.642,A 0.000,B 0.000,C 90.000,E1 295.463} C_DIS
LIN {X 0.062,Y -354.548,Z 1439.634,A 0.000,B 0.000,C 90.000,E1 294.079} C_DIS
LIN {X -0.050,Y -367.950,Z 1439.626,A 0.000,B 0.000,C 90.000,E1 292.717} C_DIS
LIN {X 0.223,Y -378.182,Z 1439.620,A 0.000,B 0.000,C 90.000,E1 291.589} C_DIS
LIN {X 0.116,Y -388.518,Z 1439.614,A 0.000,B 0.000,C 90.000,E1 290.482} C_DIS
LIN {X -0.011,Y -401.117,Z 1439.606,A 0.000,B 0.000,C 90.000,E1 289.087} C_DIS
LIN {X 0.010,Y -413.499,Z 1439.598,A 0.000,B 0.000,C 90.000,E1 287.692} C_DIS
LIN {X 0.137,Y -420.578,Z 1439.594,A 0.000,B 0.000,C 90.000,E1 286.858} C_DIS
LIN {X -0.082,Y -427.062,Z 1439.589,A 0.000,B 0.000,C 90.000,E1 286.079} C_DIS
LIN {X 0.112,Y -432.692,Z 1439.585,A 0.000,B 0.000,C 90.000,E1 285.245} C_DIS
LIN {X 0.056,Y -435.947,Z 1439.582,A 0.000,B 0.000,C 90.000,E1 284.717} C_DIS
LIN {X -0.097,Y -440.050,Z 1439.577,A 0.000,B 0.000,C 90.000,E1 283.939} C_DIS
LIN {X -0.106,Y -442.353,Z 1439.574,A 0.000,B 0.000,C 90.000,E1 283.411} C_DIS
LIN {X -0.102,Y -444.334,Z 1439.572,A 0.000,B 0.000,C 90.000,E1 282.883} C_DIS
LIN {X -0.088,Y -446.013,Z 1439.569,A 0.000,B 0.000,C 90.000,E1 282.355} C_DIS
LIN {X -0.064,Y -447.367,Z 1439.566,A 0.000,B 0.000,C 90.000,E1 281.827} C_DIS
LIN {X -0.031,Y -448.328,Z 1439.563,A 0.000,B 0.000,C 90.000,E1 281.299} C_DIS
LIN {X -0.074,Y -448.861,Z 1439.560,A 0.000,B 0.000,C 90.000,E1 280.782} C_DIS
LIN {X -0.027,Y -448.973,Z 1439.557,A 0.000,B 0.000,C 90.000,E1 280.254} C_DIS
LIN {X 0.020,Y -448.584,Z 1439.554,A 0.000,B 0.000,C 90.000,E1 279.726} C_DIS
LIN {X -0.007,Y -447.650,Z 1439.551,A 0.000,B 0.000,C 90.000,E1 279.208} C_DIS
LIN {X 0.035,Y -446.156,Z 1439.548,A 0.000,B 0.000,C 90.000,E1 278.681} C_DIS
LIN {X 0.002,Y -443.986,Z 1439.545,A 0.000,B 0.000,C 90.000,E1 278.163} C_DIS
LIN {X 0.233,Y -442.636,Z 1439.544,A 0.000,B 0.000,C 90.000,E1 277.871} C_DIS
LIN {X 0.181,Y -439.255,Z 1439.541,A 0.000,B 0.000,C 90.000,E1 277.352} C_DIS
LIN {X 0.113,Y -434.864,Z 1439.538,A 0.000,B 0.000,C 90.000,E1 276.834} C_DIS
LIN {X -0.164,Y -432.280,Z 1439.537,A 0.000,B 0.000,C 90.000,E1 276.606} C_DIS
LIN {X -0.153,Y -426.239,Z 1439.534,A 0.000,B 0.000,C 90.000,E1 276.087} C_DIS
LIN {X -0.030,Y -419.841,Z 1439.531,A 0.000,B 0.000,C 90.000,E1 275.625} C_DIS
LIN {X 0.095,Y -413.274,Z 1439.529,A 0.000,B 0.000,C 90.000,E1 275.220} C_DIS
LIN {X 0.173,Y -406.868,Z 1439.527,A 0.000,B 0.000,C 90.000,E1 274.878} C_DIS
LIN {X -0.047,Y -397.143,Z 1439.525,A 0.000,B 0.000,C 90.000,E1 274.473} C_DIS
LIN {X -0.033,Y -384.169,Z 1439.522,A 0.000,B 0.000,C 90.000,E1 273.955} C_DIS
LIN {X -0.075,Y -371.347,Z 1439.519,A 0.000,B 0.000,C 90.000,E1 273.498} C_DIS
LIN {X -0.164,Y -358.233,Z 1439.517,A 0.000,B 0.000,C 90.000,E1 273.094} C_DIS
LIN {X -0.117,Y -347.629,Z 1439.516,A 0.000,B 0.000,C 90.000,E1 272.808} C_DIS
LIN {X -0.116,Y -336.487,Z 1439.514,A 0.000,B 0.000,C 90.000,E1 272.579} C_DIS
LIN {X 0.137,Y -328.376,Z 1439.514,A 0.000,B 0.000,C 90.000,E1 272.407} C_DIS
LIN {X -0.145,Y -319.273,Z 1439.513,A 0.000,B 0.000,C 90.000,E1 272.350} C_DIS
LIN {X 0.005,Y -304.955,Z 1439.512,A 0.000,B 0.000,C 90.000,E1 272.236} C_DIS
LIN {X -0.046,Y -298.330,Z 1439.512,A 0.000,B 0.000,C 90.000,E1 272.236} C_DIS
LIN {X -0.059,Y -181.228,Z 1439.512,A 0.000,B 0.000,C 90.000,E1 272.236} C_DIS
LIN {X 0.016,Y -181.579,Z 1439.501,A 0.000,B 0.000,C 90.000,E1 270.172} C_DIS
LIN {X 0.005,Y -180.886,Z 1439.473,A 0.000,B 0.000,C 90.000,E1 265.122} C_DIS
LIN {X 0.065,Y -179.006,Z 1439.445,A 0.000,B 0.000,C 90.000,E1 260.038} C_DIS
LIN {X -0.017,Y -178.615,Z 1439.440,A 0.000,B 0.000,C 90.000,E1 259.218} C_DIS
LIN {X 0.051,Y -175.667,Z 1439.412,A 0.000,B 0.000,C 90.000,E1 254.102} C_DIS
LIN {X 0.056,Y -172.385,Z 1439.388,A 0.000,B 0.000,C 90.000,E1 249.826} C_DIS
LIN {X 0.070,Y -171.185,Z 1439.379,A 0.000,B 0.000,C 90.000,E1 248.103} C_DIS
LIN {X -0.038,Y -167.477,Z 1439.354,A 0.000,B 0.000,C 90.000,E1 243.819} C_DIS
LIN {X -0.030,Y -166.874,Z 1439.350,A 0.000,B 0.000,C 90.000,E1 242.948} C_DIS
LIN {X -0.038,Y -162.179,Z 1439.321,A 0.000,B 0.000,C 90.000,E1 237.709} C_DIS
LIN {X 0.020,Y -160.744,Z 1439.311,A 0.000,B 0.000,C 90.000,E1 235.928} C_DIS
LIN {X -0.002,Y -157.545,Z 1439.291,A 0.000,B 0.000,C 90.000,E1 232.396} C_DIS
LIN {X -0.063,Y -155.573,Z 1439.276,A 0.000,B 0.000,C 90.000,E1 229.747} C_DIS
LIN {X -0.011,Y -151.860,Z 1439.251,A 0.000,B 0.000,C 90.000,E1 225.243} C_DIS
LIN {X 0.003,Y -150.082,Z 1439.236,A 0.000,B 0.000,C 90.000,E1 222.528} C_DIS
LIN {X 0.037,Y -146.885,Z 1439.211,A 0.000,B 0.000,C 90.000,E1 217.971} C_DIS
LIN {X 0.025,Y -145.472,Z 1439.196,A 0.000,B 0.000,C 90.000,E1 215.231} C_DIS
LIN {X -0.057,Y -142.883,Z 1439.170,A 0.000,B 0.000,C 90.000,E1 210.669} C_DIS
LIN {X -0.001,Y -141.502,Z 1439.150,A 0.000,B 0.000,C 90.000,E1 206.950} C_DIS
LIN {X 0.049,Y -139.389,Z 1439.114,A 0.000,B 0.000,C 90.000,E1 200.429} C_DIS
LIN {X -0.032,Y -139.095,Z 1439.103,A 0.000,B 0.000,C 90.000,E1 198.598} C_DIS
LIN {X -0.039,Y -138.353,Z 1439.057,A 0.000,B 0.000,C 90.000,E1 190.197} C_DIS
LIN {X -0.047,Y -139.517,Z 1439.005,A 0.000,B 0.000,C 90.000,E1 180.859} C_DIS
LIN {X 0.034,Y -141.172,Z 1438.974,A 0.000,B 0.000,C 90.000,E1 175.241} C_DIS
LIN {X 0.005,Y -142.551,Z 1438.958,A 0.000,B 0.000,C 90.000,E1 172.470} C_DIS
LIN {X -0.070,Y -144.827,Z 1438.932,A 0.000,B 0.000,C 90.000,E1 167.881} C_DIS
LIN {X 0.059,Y -147.450,Z 1438.912,A 0.000,B 0.000,C 90.000,E1 164.157} C_DIS
LIN {X -0.055,Y -150.031,Z 1438.892,A 0.000,B 0.000,C 90.000,E1 160.550} C_DIS
LIN {X -0.049,Y -153.369,Z 1438.872,A 0.000,B 0.000,C 90.000,E1 156.922} C_DIS
LIN {X 0.000,Y -155.902,Z 1438.857,A 0.000,B 0.000,C 90.000,E1 154.204} C_DIS
LIN {X -0.025,Y -159.763,Z 1438.837,A 0.000,B 0.000,C 90.000,E1 150.639} C_DIS
LIN {X -0.037,Y -162.002,Z 1438.827,A 0.000,B 0.000,C 90.000,E1 148.869} C_DIS
LIN {X 0.077,Y -166.196,Z 1438.807,A 0.000,B 0.000,C 90.000,E1 145.308} C_DIS
LIN {X 0.079,Y -171.211,Z 1438.788,A 0.000,B 0.000,C 90.000,E1 141.823} C_DIS
LIN {X 0.004,Y -176.096,Z 1438.769,A 0.000,B 0.000,C 90.000,E1 138.405} C_DIS
LIN {X -0.005,Y -180.357,Z 1438.755,A 0.000,B 0.000,C 90.000,E1 135.850} C_DIS
LIN {X 0.098,Y -185.767,Z 1438.736,A 0.000,B 0.000,C 90.000,E1 132.447} C_DIS
LIN {X 0.031,Y -190.380,Z 1438.722,A 0.000,B 0.000,C 90.000,E1 129.967} C_DIS
LIN {X -0.069,Y -197.705,Z 1438.699,A 0.000,B 0.000,C 90.000,E1 125.884} C_DIS
LIN {X -0.001,Y -200.340,Z 1438.692,A 0.000,B 0.000,C 90.000,E1 124.565} C_DIS
LIN {X 0.123,Y -311.829,Z 1438.692,A 0.000,B 0.000,C 90.000,E1 124.532} C_DIS
LIN {X -0.076,Y -317.024,Z 1438.691,A 0.000,B 0.000,C 90.000,E1 124.405} C_DIS
LIN {X -0.044,Y -319.280,Z 1438.690,A 0.000,B 0.000,C 90.000,E1 124.246} C_DIS
LIN {X -0.008,Y -323.146,Z 1438.688,A 0.000,B 0.000,C 90.000,E1 123.833} C_DIS
LIN {X -0.211,Y -325.051,Z 1438.686,A 0.000,B 0.000,C 90.000,E1 123.579} C_DIS
LIN {X 0.039,Y -326.549,Z 1438.685,A 0.000,B 0.000,C 90.000,E1 123.245} C_DIS
LIN {X -0.036,Y -328.961,Z 1438.681,A 0.000,B 0.000,C 90.000,E1 122.625} C_DIS
LIN {X 0.050,Y -339.706,Z 1438.666,A 0.000,B 0.000,C 90.000,E1 119.795} C_DIS
LIN {X -0.076,Y -351.818,Z 1438.650,A 0.000,B 0.000,C 90.000,E1 117.052} C_DIS
LIN {X -0.011,Y -365.394,Z 1438.635,A 0.000,B 0.000,C 90.000,E1 114.335} C_DIS
LIN {X 0.041,Y -378.789,Z 1438.622,A 0.000,B 0.000,C 90.000,E1 111.972} C_DIS
LIN {X -0.074,Y -393.531,Z 1438.609,A 0.000,B 0.000,C 90.000,E1 109.685} C_DIS
LIN {X 0.150,Y -409.720,Z 1438.597,A 0.000,B 0.000,C 90.000,E1 107.402} C_DIS
LIN {X -0.128,Y -427.470,Z 1438.585,A 0.000,B 0.000,C 90.000,E1 105.245} C_DIS
LIN {X -0.146,Y -446.815,Z 1438.573,A 0.000,B 0.000,C 90.000,E1 103.119} C_DIS
LIN {X -0.053,Y -466.981,Z 1438.562,A 0.000,B 0.000,C 90.000,E1 101.130} C_DIS
LIN {X -0.122,Y -487.504,Z 1438.552,A 0.000,B 0.000,C 90.000,E1 99.321} C_DIS
LIN {X -0.050,Y -489.359,Z 1438.551,A 0.000,B 0.000,C 90.000,E1 99.095} C_DIS
LIN {X -0.151,Y -490.956,Z 1438.549,A 0.000,B 0.000,C 90.000,E1 98.859} C_DIS
LIN {X 0.232,Y -492.150,Z 1438.548,A 0.000,B 0.000,C 90.000,E1 98.568} C_DIS
LIN {X -0.028,Y -493.585,Z 1438.545,A 0.000,B 0.000,C 90.000,E1 98.106} C_DIS
LIN {X 0.208,Y -493.967,Z 1438.542,A 0.000,B 0.000,C 90.000,E1 97.587} C_DIS
LIN {X -0.036,Y -493.358,Z 1438.540,A 0.000,B 0.000,C 90.000,E1 97.125} C_DIS
LIN {X 0.212,Y -491.662,Z 1438.537,A 0.000,B 0.000,C 90.000,E1 96.606} C_DIS
LIN {X 0.116,Y -490.309,Z 1438.536,A 0.000,B 0.000,C 90.000,E1 96.372} C_DIS
LIN {X -0.085,Y -477.058,Z 1438.525,A 0.000,B 0.000,C 90.000,E1 94.416} C_DIS
LIN {X -0.196,Y -467.735,Z 1438.516,A 0.000,B 0.000,C 90.000,E1 92.922} C_DIS
LIN {X 0.190,Y -459.477,Z 1438.509,A 0.000,B 0.000,C 90.000,E1 91.604} C_DIS
LIN {X 0.162,Y -445.966,Z 1438.498,A 0.000,B 0.000,C 90.000,E1 89.542} C_DIS
LIN {X -0.005,Y -431.354,Z 1438.484,A 0.000,B 0.000,C 90.000,E1 87.192} C_DIS
LIN {X 0.107,Y -419.980,Z 1438.474,A 0.000,B 0.000,C 90.000,E1 85.298} C_DIS
LIN {X -0.058,Y -410.207,Z 1438.465,A 0.000,B 0.000,C 90.000,E1 83.685} C_DIS
LIN {X 0.095,Y -398.709,Z 1438.454,A 0.000,B 0.000,C 90.000,E1 81.724} C_DIS
LIN {X 0.123,Y -387.030,Z 1438.443,A 0.000,B 0.000,C 90.000,E1 79.746} C_DIS
LIN {X 0.012,Y -370.565,Z 1438.427,A 0.000,B 0.000,C 90.000,E1 76.881} C_DIS
LIN {X 0.061,Y -359.287,Z 1438.416,A 0.000,B 0.000,C 90.000,E1 74.810} C_DIS
LIN {X 0.041,Y -349.558,Z 1438.406,A 0.000,B 0.000,C 90.000,E1 73.015} C_DIS
LIN {X -0.148,Y -338.019,Z 1438.394,A 0.000,B 0.000,C 90.000,E1 70.913} C_DIS
LIN {X -0.082,Y -325.043,Z 1438.380,A 0.000,B 0.000,C 90.000,E1 68.411} C_DIS
LIN {X -0.050,Y -311.012,Z 1438.364,A 0.000,B 0.000,C 90.000,E1 65.537} C_DIS
LIN {X -0.133,Y -298.141,Z 1438.348,A 0.000,B 0.000,C 90.000,E1 62.615} C_DIS
LIN {X -0.035,Y -285.200,Z 1438.329,A 0.000,B 0.000,C 90.000,E1 59.253} C_DIS
LIN {X 0.103,Y -273.351,Z 1438.310,A 0.000,B 0.000,C 90.000,E1 55.801} C_DIS
LIN {X -0.027,Y -263.217,Z 1438.293,A 0.000,B 0.000,C 90.000,E1 52.683} C_DIS
LIN {X 0.065,Y -253.757,Z 1438.275,A 0.000,B 0.000,C 90.000,E1 49.461} C_DIS
LIN {X 0.006,Y -244.175,Z 1438.255,A 0.000,B 0.000,C 90.000,E1 45.850} C_DIS
LIN {X -0.012,Y -235.442,Z 1438.234,A 0.000,B 0.000,C 90.000,E1 42.162} C_DIS
LIN {X 0.075,Y -227.574,Z 1438.213,A 0.000,B 0.000,C 90.000,E1 38.382} C_DIS
LIN {X -0.108,Y -220.574,Z 1438.192,A 0.000,B 0.000,C 90.000,E1 34.612} C_DIS
LIN {X -0.028,Y -214.402,Z 1438.171,A 0.000,B 0.000,C 90.000,E1 30.718} C_DIS
LIN {X -0.028,Y -208.975,Z 1438.149,A 0.000,B 0.000,C 90.000,E1 26.796} C_DIS
LIN {X -0.007,Y -204.407,Z 1438.127,A 0.000,B 0.000,C 90.000,E1 22.823} C_DIS
LIN {X 0.035,Y -200.021,Z 1438.100,A 0.000,B 0.000,C 90.000,E1 18.000} C_DIS
LIN {X -0.040,Y -196.274,Z 1438.069,A 0.000,B 0.000,C 90.000,E1 12.355} C_DIS
LIN {X -0.048,Y -194.014,Z 1438.041,A 0.000,B 0.000,C 90.000,E1 7.466} C_DIS
LIN {X -0.086,Y -192.777,Z 1438.019,A 0.000,B 0.000,C 90.000,E1 3.383} C_DIS
LIN {X 0.091,Y -192.035,Z 1437.993,A 0.000,B 0.000,C 90.000,E1 358.682} C_DIS
LIN {X -0.073,Y -191.915,Z 1437.965,A 0.000,B 0.000,C 90.000,E1 353.799} C_DIS
LIN {X -0.084,Y -192.649,Z 1437.933,A 0.000,B 0.000,C 90.000,E1 348.049} C_DIS
LIN {X 0.039,Y -195.303,Z 1437.897,A 0.000,B 0.000,C 90.000,E1 341.456} C_DIS
LIN {X -0.112,Y -198.852,Z 1437.870,A 0.000,B 0.000,C 90.000,E1 336.613} C_DIS
LIN {X 0.008,Y -202.998,Z 1437.847,A 0.000,B 0.000,C 90.000,E1 332.538} C_DIS
LIN {X 0.010,Y -208.246,Z 1437.825,A 0.000,B 0.000,C 90.000,E1 328.535} C_DIS
LIN {X -0.069,Y -213.372,Z 1437.808,A 0.000,B 0.000,C 90.000,E1 325.388} C_DIS
LIN {X -0.129,Y -219.520,Z 1437.790,A 0.000,B 0.000,C 90.000,E1 322.271} C_DIS
LIN {X 0.033,Y -226.654,Z 1437.773,A 0.000,B 0.000,C 90.000,E1 319.138} C_DIS
LIN {X -0.002,Y -235.782,Z 1437.754,A 0.000,B 0.000,C 90.000,E1 315.729} C_DIS
LIN {X -0.097,Y -244.858,Z 1437.738,A 0.000,B 0.000,C 90.000,E1 312.771} C_DIS
LIN {X -0.097,Y -256.312,Z 1437.719,A 0.000,B 0.000,C 90.000,E1 309.483} C_DIS
LIN {X 0.034,Y -266.240,Z 1437.705,A 0.000,B 0.000,C 90.000,E1 306.950} C_DIS
LIN {X 0.151,Y -275.731,Z 1437.694,A 0.000,B 0.000,C 90.000,E1 304.818} C_DIS
LIN {X 0.139,Y -286.226,Z 1437.682,A 0.000,B 0.000,C 90.000,E1 302.752} C_DIS
LIN {X 0.023,Y -296.177,Z 1437.673,A 0.000,B 0.000,C 90.000,E1 301.082} C_DIS
LIN {X 0.047,Y -304.900,Z 1437.665,A 0.000,B 0.000,C 90.000,E1 299.745} C_DIS
LIN {X 0.138,Y -312.084,Z 1437.660,A 0.000,B 0.000,C 90.000,E1 298.743} C_DIS
LIN {X 0.074,Y -327.348,Z 1437.650,A 0.000,B 0.000,C 90.000,E1 296.924} C_DIS
LIN {X 0.155,Y -349.022,Z 1437.637,A 0.000,B 0.000,C 90.000,E1 294.643} C_DIS
LIN {X -0.014,Y -359.849,Z 1437.631,A 0.000,B 0.000,C 90.000,E1 293.567} C_DIS
LIN {X 0.016,Y -370.474,Z 1437.625,A 0.000,B 0.000,C 90.000,E1 292.461} C_DIS
LIN {X -0.029,Y -380.844,Z 1437.619,A 0.000,B 0.000,C 90.000,E1 291.354} C_DIS
LIN {X -0.061,Y -390.972,Z 1437.612,A 0.000,B 0.000,C 90.000,E1 290.248} C_DIS
LIN {X 0.176,Y -401.001,Z 1437.606,A 0.000,B 0.000,C 90.000,E1 289.087} C_DIS
LIN {X -0.123,Y -415.891,Z 1437.597,A 0.000,B 0.000,C 90.000,E1 287.457} C_DIS
LIN {X -0.042,Y -422.901,Z 1437.592,A 0.000,B 0.000,C 90.000,E1 286.622} C_DIS
LIN {X -0.044,Y -427.191,Z 1437.589,A 0.000,B 0.000,C 90.000,E1 286.079} C_DIS
LIN {X 0.151,Y -432.864,Z 1437.585,A 0.000,B 0.000,C 90.000,E1 285.245} C_DIS
LIN {X -0.137,Y -437.561,Z 1437.580,A 0.000,B 0.000,C 90.000,E1 284.481} C_DIS
LIN {X 0.156,Y -441.422,Z 1437.576,A 0.000,B 0.000,C 90.000,E1 283.647} C_DIS
LIN {X -0.056,Y -444.531,Z 1437.572,A 0.000,B 0.000,C 90.000,E1 282.883} C_DIS
LIN {X -0.042,Y -446.235,Z 1437.569,A 0.000,B 0.000,C 90.000,E1 282.355} C_DIS
LIN {X -0.016,Y -447.590,Z 1437.566,A 0.000,B 0.000,C 90.000,E1 281.827} C_DIS
LIN {X 0.019,Y -448.590,Z 1437.563,A 0.000,B 0.000,C 90.000,E1 281.299} C_DIS
LIN {X -0.024,Y -449.158,Z 1437.560,A 0.000,B 0.000,C 90.000,E1 280.782} C_DIS
LIN {X 0.025,Y -449.264,Z 1437.557,A 0.000,B 0.000,C 90.000,E1 280.254} C_DIS
LIN {X 0.074,Y -448.944,Z 1437.554,A 0.000,B 0.000,C 90.000,E1 279.726} C_DIS
LIN {X 0.048,Y -448.026,Z 1437.551,A 0.000,B 0.000,C 90.000,E1 279.208} C_DIS
LIN {X 0.091,Y -446.547,Z 1437.548,A 0.000,B 0.000,C 90.000,E1 278.681} C_DIS
LIN {X 0.061,Y -444.409,Z 1437.545,A 0.000,B 0.000,C 90.000,E1 278.163} C_DIS
LIN {X 0.025,Y -441.531,Z 1437.542,A 0.000,B 0.000,C 90.000,E1 277.644} C_DIS
LIN {X -0.030,Y -437.752,Z 1437.540,A 0.000,B 0.000,C 90.000,E1 277.125} C_DIS
LIN {X -0.100,Y -432.866,Z 1437.537,A 0.000,B 0.000,C 90.000,E1 276.606} C_DIS
LIN {X 0.140,Y -430.060,Z 1437.535,A 0.000,B 0.000,C 90.000,E1 276.315} C_DIS
LIN {X 0.003,Y -423.877,Z 1437.532,A 0.000,B 0.000,C 90.000,E1 275.853} C_DIS
LIN {X -0.090,Y -417.528,Z 1437.530,A 0.000,B 0.000,C 90.000,E1 275.448} C_DIS
LIN {X 0.153,Y -410.972,Z 1437.528,A 0.000,B 0.000,C 90.000,E1 275.049} C_DIS
LIN {X 0.085,Y -401.079,Z 1437.526,A 0.000,B 0.000,C 90.000,E1 274.588} C_DIS
LIN {X 0.075,Y -391.450,Z 1437.523,A 0.000,B 0.000,C 90.000,E1 274.188} C_DIS
LIN {X -0.089,Y -378.675,Z 1437.521,A 0.000,B 0.000,C 90.000,E1 273.726} C_DIS
LIN {X -0.028,Y -365.595,Z 1437.518,A 0.000,B 0.000,C 90.000,E1 273.269} C_DIS
LIN {X -0.104,Y -355.484,Z 1437.516,A 0.000,B 0.000,C 90.000,E1 272.980} C_DIS
LIN {X 0.082,Y -344.903,Z 1437.515,A 0.000,B 0.000,C 90.000,E1 272.694} C_DIS
LIN {X 0.155,Y -333.429,Z 1437.514,A 0.000,B 0.000,C 90.000,E1 272.465} C_DIS
LIN {X -0.137,Y -320.195,Z 1437.513,A 0.000,B 0.000,C 90.000,E1 272.350} C_DIS
LIN {X 0.116,Y -310.596,Z 1437.513,A 0.000,B 0.000,C 90.000,E1 272.236} C_DIS
LIN {X 0.007,Y -305.386,Z 1437.512,A 0.000,B 0.000,C 90.000,E1 272.236} C_DIS
LIN {X -0.028,Y -181.226,Z 1437.512,A 0.000,B 0.000,C 90.000,E1 272.236} C_DIS
LIN {X -0.010,Y -181.563,Z 1437.503,A 0.000,B 0.000,C 90.000,E1 270.516} C_DIS
LIN {X -0.081,Y -181.281,Z 1437.494,A 0.000,B 0.000,C 90.000,E1 268.854} C_DIS
LIN {X -0.032,Y -180.907,Z 1437.475,A 0.000,B 0.000,C 90.000,E1 265.469} C_DIS
LIN {X 0.025,Y -180.732,Z 1437.470,A 0.000,B 0.000,C 90.000,E1 264.609} C_DIS
LIN {X -0.054,Y -178.821,Z 1437.442,A 0.000,B 0.000,C 90.000,E1 259.567} C_DIS
LIN {X 0.028,Y -175.866,Z 1437.414,A 0.000,B 0.000,C 90.000,E1 254.448} C_DIS
LIN {X 0.022,Y -173.835,Z 1437.399,A 0.000,B 0.000,C 90.000,E1 251.891} C_DIS
LIN {X 0.012,Y -171.502,Z 1437.380,A 0.000,B 0.000,C 90.000,E1 248.465} C_DIS
LIN {X -0.001,Y -167.730,Z 1437.356,A 0.000,B 0.000,C 90.000,E1 244.152} C_DIS
LIN {X 0.014,Y -166.426,Z 1437.347,A 0.000,B 0.000,C 90.000,E1 242.410} C_DIS
LIN {X 0.013,Y -163.147,Z 1437.327,A 0.000,B 0.000,C 90.000,E1 238.918} C_DIS
LIN {X -0.021,Y -161.102,Z 1437.313,A 0.000,B 0.000,C 90.000,E1 236.294} C_DIS
LIN {X -0.038,Y -157.829,Z 1437.293,A 0.000,B 0.000,C 90.000,E1 232.763} C_DIS
LIN {X 0.025,Y -155.863,Z 1437.278,A 0.000,B 0.000,C 90.000,E1 230.070} C_DIS
LIN {X 0.081,Y -152.113,Z 1437.253,A 0.000,B 0.000,C 90.000,E1 225.567} C_DIS
LIN {X -0.011,Y -150.363,Z 1437.238,A 0.000,B 0.000,C 90.000,E1 222.894} C_DIS
LIN {X 0.027,Y -147.098,Z 1437.213,A 0.000,B 0.000,C 90.000,E1 218.338} C_DIS
LIN {X 0.022,Y -145.667,Z 1437.198,A 0.000,B 0.000,C 90.000,E1 215.598} C_DIS
LIN {X 0.025,Y -143.050,Z 1437.172,A 0.000,B 0.000,C 90.000,E1 211.003} C_DIS
LIN {X -0.039,Y -141.673,Z 1437.152,A 0.000,B 0.000,C 90.000,E1 207.334} C_DIS
LIN {X 0.070,Y -139.454,Z 1437.116,A 0.000,B 0.000,C 90.000,E1 200.791} C_DIS
LIN {X -0.010,Y -139.187,Z 1437.105,A 0.000,B 0.000,C 90.000,E1 198.960} C_DIS
LIN {X 0.013,Y -138.323,Z 1437.053,A 0.000,B 0.000,C 90.000,E1 189.613} C_DIS
LIN {X 0.020,Y -139.459,Z 1437.007,A 0.000,B 0.000,C 90.000,E1 181.203} C_DIS
LIN {X -0.039,Y -141.014,Z 1436.976,A 0.000,B 0.000,C 90.000,E1 175.641} C_DIS
LIN {X 0.051,Y -142.767,Z 1436.955,A 0.000,B 0.000,C 90.000,E1 171.894} C_DIS
LIN {X 0.007,Y -145.177,Z 1436.929,A 0.000,B 0.000,C 90.000,E1 167.297} C_DIS
LIN {X 0.040,Y -147.799,Z 1436.909,A 0.000,B 0.000,C 90.000,E1 163.614} C_DIS
LIN {X -0.065,Y -150.483,Z 1436.889,A 0.000,B 0.000,C 90.000,E1 160.007} C_DIS
LIN {X 0.008,Y -153.938,Z 1436.869,A 0.000,B 0.000,C 90.000,E1 156.357} C_DIS
LIN {X 0.071,Y -157.349,Z 1436.849,A 0.000,B 0.000,C 90.000,E1 152.743} C_DIS
LIN {X 0.015,Y -161.545,Z 1436.829,A 0.000,B 0.000,C 90.000,E1 149.203} C_DIS
LIN {X 0.028,Y -165.743,Z 1436.809,A 0.000,B 0.000,C 90.000,E1 145.674} C_DIS
LIN {X 0.015,Y -170.696,Z 1436.790,A 0.000,B 0.000,C 90.000,E1 142.190} C_DIS
LIN {X -0.074,Y -175.570,Z 1436.771,A 0.000,B 0.000,C 90.000,E1 138.771} C_DIS
LIN {X 0.045,Y -181.188,Z 1436.752,A 0.000,B 0.000,C 90.000,E1 135.324} C_DIS
LIN {X -0.086,Y -186.648,Z 1436.733,A 0.000,B 0.000,C 90.000,E1 132.000} C_DIS
LIN {X -0.017,Y -191.253,Z 1436.719,A 0.000,B 0.000,C 90.000,E1 129.483} C_DIS
LIN {X 0.064,Y -197.073,Z 1436.701,A 0.000,B 0.000,C 90.000,E1 126.171} C_DIS
LIN {X -0.106,Y -200.305,Z 1436.692,A 0.000,B 0.000,C 90.000,E1 124.612} C_DIS
LIN {X 0.037,Y -312.303,Z 1436.692,A 0.000,B 0.000,C 90.000,E1 124.565} C_DIS
LIN {X -0.032,Y -316.306,Z 1436.691,A 0.000,B 0.000,C 90.000,E1 124.452} C_DIS
LIN {X -0.080,Y -319.530,Z 1436.690,A 0.000,B 0.000,C 90.000,E1 124.246} C_DIS
LIN {X -0.007,Y -323.209,Z 1436.688,A 0.000,B 0.000,C 90.000,E1 123.833} C_DIS
LIN {X 0.202,Y -325.118,Z 1436.686,A 0.000,B 0.000,C 90.000,E1 123.499} C_DIS
LIN {X -0.039,Y -326.614,Z 1436.685,A 0.000,B 0.000,C 90.000,E1 123.245} C_DIS
LIN {X -0.176,Y -331.265,Z 1436.678,A 0.000,B 0.000,C 90.000,E1 122.005} C_DIS
LIN {X 0.095,Y -342.311,Z 1436.662,A 0.000,B 0.000,C 90.000,E1 119.155} C_DIS
LIN {X 0.050,Y -354.745,Z 1436.647,A 0.000,B 0.000,C 90.000,E1 116.411} C_DIS
LIN {X 0.054,Y -368.670,Z 1436.632,A 0.000,B 0.000,C 90.000,E1 113.718} C_DIS
LIN {X -0.158,Y -382.401,Z 1436.619,A 0.000,B 0.000,C 90.000,E1 111.408} C_DIS
LIN {X 0.041,Y -397.502,Z 1436.606,A 0.000,B 0.000,C 90.000,E1 109.087} C_DIS
LIN {X -0.016,Y -414.079,Z 1436.594,A 0.000,B 0.000,C 90.000,E1 106.858} C_DIS
LIN {X 0.105,Y -432.247,Z 1436.582,A 0.000,B 0.000,C 90.000,E1 104.662} C_DIS
LIN {X -0.096,Y -451.890,Z 1436.570,A 0.000,B 0.000,C 90.000,E1 102.591} C_DIS
LIN {X -0.117,Y -472.198,Z 1436.559,A 0.000,B 0.000,C 90.000,E1 100.658} C_DIS
LIN {X 0.120,Y -485.167,Z 1436.553,A 0.000,B 0.000,C 90.000,E1 99.500} C_DIS
LIN {X -0.209,Y -487.554,Z 1436.552,A 0.000,B 0.000,C 90.000,E1 99.321} C_DIS
LIN {X -0.137,Y -489.366,Z 1436.550,A 0.000,B 0.000,C 90.000,E1 99.095} C_DIS
LIN {X -0.238,Y -490.930,Z 1436.549,A 0.000,B 0.000,C 90.000,E1 98.859} C_DIS
LIN {X 0.145,Y -492.096,Z 1436.548,A 0.000,B 0.000,C 90.000,E1 98.568} C_DIS
LIN {X -0.116,Y -493.490,Z 1436.545,A 0.000,B 0.000,C 90.000,E1 98.106} C_DIS
LIN {X 0.120,Y -493.835,Z 1436.542,A 0.000,B 0.000,C 90.000,E1 97.587} C_DIS
LIN {X -0.125,Y -493.190,Z 1436.540,A 0.000,B 0.000,C 90.000,E1 97.125} C_DIS
LIN {X 0.123,Y -491.450,Z 1436.537,A 0.000,B 0.000,C 90.000,E1 96.606} C_DIS
LIN {X 0.027,Y -490.068,Z 1436.535,A 0.000,B 0.000,C 90.000,E1 96.372} C_DIS
LIN {X -0.176,Y -476.826,Z 1436.524,A 0.000,B 0.000,C 90.000,E1 94.416} C_DIS
LIN {X -0.118,Y -469.091,Z 1436.517,A 0.000,B 0.000,C 90.000,E1 93.154} C_DIS
LIN {X -0.169,Y -460.887,Z 1436.510,A 0.000,B 0.000,C 90.000,E1 91.892} C_DIS
LIN {X -0.143,Y -447.381,Z 1436.499,A 0.000,B 0.000,C 90.000,E1 89.828} C_DIS
LIN {X -0.106,Y -431.155,Z 1436.484,A 0.000,B 0.000,C 90.000,E1 87.192} C_DIS
LIN {X 0.005,Y -419.806,Z 1436.474,A 0.000,B 0.000,C 90.000,E1 85.298} C_DIS
LIN {X -0.161,Y -410.045,Z 1436.465,A 0.000,B 0.000,C 90.000,E1 83.685} C_DIS
LIN {X -0.008,Y -398.609,Z 1436.454,A 0.000,B 0.000,C 90.000,E1 81.724} C_DIS
LIN {X 0.021,Y -386.929,Z 1436.443,A 0.000,B 0.000,C 90.000,E1 79.746} C_DIS
LIN {X -0.095,Y -372.090,Z 1436.429,A 0.000,B 0.000,C 90.000,E1 77.173} C_DIS
LIN {X -0.003,Y -360.813,Z 1436.417,A 0.000,B 0.000,C 90.000,E1 75.102} C_DIS
LIN {X -0.091,Y -351.109,Z 1436.407,A 0.000,B 0.000,C 90.000,E1 73.323} C_DIS
LIN {X 0.173,Y -341.235,Z 1436.397,A 0.000,B 0.000,C 90.000,E1 71.456} C_DIS
LIN {X -0.116,Y -328.159,Z 1436.383,A 0.000,B 0.000,C 90.000,E1 69.028} C_DIS
LIN {X -0.126,Y -313.948,Z 1436.368,A 0.000,B 0.000,C 90.000,E1 66.177} C_DIS
LIN {X -0.025,Y -302.159,Z 1436.353,A 0.000,B 0.000,C 90.000,E1 63.563} C_DIS
LIN {X -0.085,Y -288.840,Z 1436.335,A 0.000,B 0.000,C 90.000,E1 60.255} C_DIS
LIN {X 0.019,Y -276.738,Z 1436.316,A 0.000,B 0.000,C 90.000,E1 56.834} C_DIS
LIN {X 0.048,Y -266.498,Z 1436.298,A 0.000,B 0.000,C 90.000,E1 53.703} C_DIS
LIN {X -0.093,Y -255.806,Z 1436.279,A 0.000,B 0.000,C 90.000,E1 50.194} C_DIS
LIN {X 0.105,Y -246.052,Z 1436.259,A 0.000,B 0.000,C 90.000,E1 46.539} C_DIS
LIN {X -0.037,Y -237.205,Z 1436.238,A 0.000,B 0.000,C 90.000,E1 42.894} C_DIS
LIN {X 0.099,Y -229.176,Z 1436.217,A 0.000,B 0.000,C 90.000,E1 39.116} C_DIS
LIN {X 0.094,Y -222.006,Z 1436.196,A 0.000,B 0.000,C 90.000,E1 35.311} C_DIS
LIN {X 0.035,Y -215.704,Z 1436.175,A 0.000,B 0.000,C 90.000,E1 31.465} C_DIS
LIN {X -0.006,Y -210.140,Z 1436.153,A 0.000,B 0.000,C 90.000,E1 27.564} C_DIS
LIN {X 0.052,Y -205.437,Z 1436.131,A 0.000,B 0.000,C 90.000,E1 23.590} C_DIS
LIN {X 0.087,Y -200.880,Z 1436.104,A 0.000,B 0.000,C 90.000,E1 18.779} C_DIS
LIN {X 0.020,Y -197.468,Z 1436.078,A 0.000,B 0.000,C 90.000,E1 13.953} C_DIS
LIN {X -0.053,Y -194.943,Z 1436.050,A 0.000,B 0.000,C 90.000,E1 9.095} C_DIS
LIN {X -0.044,Y -193.290,Z 1436.023,A 0.000,B 0.000,C 90.000,E1 4.188} C_DIS
LIN {X 0.093,Y -192.317,Z 1435.993,A 0.000,B 0.000,C 90.000,E1 358.682} C_DIS
LIN {X -0.060,Y -192.195,Z 1435.965,A 0.000,B 0.000,C 90.000,E1 353.799} C_DIS
LIN {X -0.061,Y -192.894,Z 1435.933,A 0.000,B 0.000,C 90.000,E1 348.049} C_DIS
LIN {X 0.075,Y -195.509,Z 1435.897,A 0.000,B 0.000,C 90.000,E1 341.456} C_DIS
LIN {X -0.068,Y -199.037,Z 1435.870,A 0.000,B 0.000,C 90.000,E1 336.613} C_DIS
LIN {X 0.060,Y -203.177,Z 1435.848,A 0.000,B 0.000,C 90.000,E1 332.538} C_DIS
LIN {X 0.068,Y -208.424,Z 1435.825,A 0.000,B 0.000,C 90.000,E1 328.535} C_DIS
LIN {X -0.004,Y -213.548,Z 1435.808,A 0.000,B 0.000,C 90.000,E1 325.388} C_DIS
LIN {X -0.058,Y -219.693,Z 1435.790,A 0.000,B 0.000,C 90.000,E1 322.271} C_DIS
LIN {X -0.037,Y -226.820,Z 1435.773,A 0.000,B 0.000,C 90.000,E1 319.175} C_DIS
LIN {X 0.083,Y -235.941,Z 1435.754,A 0.000,B 0.000,C 90.000,E1 315.729} C_DIS
LIN {X -0.004,Y -245.009,Z 1435.738,A 0.000,B 0.000,C 90.000,E1 312.771} C_DIS
LIN {X 0.005,Y -256.447,Z 1435.719,A 0.000,B 0.000,C 90.000,E1 309.483} C_DIS
LIN {X -0.013,Y -267.858,Z 1435.703,A 0.000,B 0.000,C 90.000,E1 306.629} C_DIS
LIN {X -0.093,Y -279.175,Z 1435.690,A 0.000,B 0.000,C 90.000,E1 304.199} C_DIS
LIN {X -0.020,Y -288.187,Z 1435.680,A 0.000,B 0.000,C 90.000,E1 302.467} C_DIS
LIN {X -0.107,Y -298.347,Z 1435.671,A 0.000,B 0.000,C 90.000,E1 300.797} C_DIS
LIN {X -0.063,Y -307.264,Z 1435.664,A 0.000,B 0.000,C 90.000,E1 299.461} C_DIS
LIN {X 0.067,Y -317.098,Z 1435.656,A 0.000,B 0.000,C 90.000,E1 298.153} C_DIS
LIN {X 0.056,Y -329.913,Z 1435.648,A 0.000,B 0.000,C 90.000,E1 296.668} C_DIS
LIN {X 0.007,Y -348.745,Z 1435.637,A 0.000,B 0.000,C 90.000,E1 294.719} C_DIS
LIN {X 0.060,Y -362.187,Z 1435.630,A 0.000,B 0.000,C 90.000,E1 293.334} C_DIS
LIN {X 0.190,Y -372.787,Z 1435.624,A 0.000,B 0.000,C 90.000,E1 292.206} C_DIS
LIN {X -0.104,Y -385.749,Z 1435.616,A 0.000,B 0.000,C 90.000,E1 290.844} C_DIS
LIN {X -0.151,Y -398.334,Z 1435.608,A 0.000,B 0.000,C 90.000,E1 289.450} C_DIS
LIN {X -0.115,Y -413.297,Z 1435.599,A 0.000,B 0.000,C 90.000,E1 287.764} C_DIS
LIN {X 0.073,Y -420.500,Z 1435.594,A 0.000,B 0.000,C 90.000,E1 286.913} C_DIS
LIN {X -0.064,Y -425.023,Z 1435.591,A 0.000,B 0.000,C 90.000,E1 286.386} C_DIS
LIN {X 0.109,Y -431.006,Z 1435.586,A 0.000,B 0.000,C 90.000,E1 285.552} C_DIS
LIN {X 0.156,Y -434.517,Z 1435.583,A 0.000,B 0.000,C 90.000,E1 285.009} C_DIS
LIN {X -0.113,Y -438.955,Z 1435.579,A 0.000,B 0.000,C 90.000,E1 284.245} C_DIS
LIN {X 0.189,Y -442.616,Z 1435.575,A 0.000,B 0.000,C 90.000,E1 283.411} C_DIS
LIN {X 0.197,Y -444.656,Z 1435.572,A 0.000,B 0.000,C 90.000,E1 282.883} C_DIS
LIN {X 0.213,Y -446.368,Z 1435.569,A 0.000,B 0.000,C 90.000,E1 282.355} C_DIS
LIN {X 0.240,Y -447.765,Z 1435.566,A 0.000,B 0.000,C 90.000,E1 281.827} C_DIS
LIN {X -0.252,Y -448.801,Z 1435.563,A 0.000,B 0.000,C 90.000,E1 281.366} C_DIS
LIN {X -0.207,Y -449.419,Z 1435.560,A 0.000,B 0.000,C 90.000,E1 280.838} C_DIS
LIN {X -0.157,Y -449.594,Z 1435.557,A 0.000,B 0.000,C 90.000,E1 280.310} C_DIS
LIN {X -0.107,Y -449.274,Z 1435.554,A 0.000,B 0.000,C 90.000,E1 279.782} C_DIS
LIN {X -0.131,Y -448.432,Z 1435.551,A 0.000,B 0.000,C 90.000,E1 279.265} C_DIS
LIN {X -0.154,Y -446.989,Z 1435.548,A 0.000,B 0.000,C 90.000,E1 278.746} C_DIS
LIN {X -0.114,Y -444.940,Z 1435.546,A 0.000,B 0.000,C 90.000,E1 278.219} C_DIS
LIN {X -0.147,Y -442.166,Z 1435.543,A 0.000,B 0.000,C 90.000,E1 277.701} C_DIS
LIN {X -0.197,Y -438.487,Z 1435.540,A 0.000,B 0.000,C 90.000,E1 277.182} C_DIS
LIN {X 0.168,Y -433.768,Z 1435.537,A 0.000,B 0.000,C 90.000,E1 276.606} C_DIS
LIN {X -0.069,Y -430.930,Z 1435.535,A 0.000,B 0.000,C 90.000,E1 276.372} C_DIS
LIN {X 0.135,Y -424.762,Z 1435.533,A 0.000,B 0.000,C 90.000,E1 275.853} C_DIS
LIN {X -0.038,Y -418.415,Z 1435.530,A 0.000,B 0.000,C 90.000,E1 275.454} C_DIS
LIN {X -0.179,Y -411.888,Z 1435.528,A 0.000,B 0.000,C 90.000,E1 275.106} C_DIS
LIN {X 0.133,Y -402.050,Z 1435.526,A 0.000,B 0.000,C 90.000,E1 274.588} C_DIS
LIN {X 0.095,Y -392.346,Z 1435.523,A 0.000,B 0.000,C 90.000,E1 274.188} C_DIS
LIN {X -0.067,Y -379.644,Z 1435.521,A 0.000,B 0.000,C 90.000,E1 273.726} C_DIS
LIN {X -0.033,Y -366.506,Z 1435.518,A 0.000,B 0.000,C 90.000,E1 273.269} C_DIS
LIN {X -0.141,Y -356.222,Z 1435.516,A 0.000,B 0.000,C 90.000,E1 272.980} C_DIS
LIN {X 0.046,Y -345.581,Z 1435.515,A 0.000,B 0.000,C 90.000,E1 272.694} C_DIS
